  PROC DrawPart187()
    MoveL Offs(pOrigin,194.96,273.17,0.00),v40,fine,tPen\WObj:=wPaper;
    MoveL Offs(pOrigin,194.96,273.17,6.00),v60,z5,tPen\WObj:=wPaper;
    MoveL Offs(pOrigin,203.82,260.21,6.00),vTravel,z5,tPen\WObj:=wPaper;
    MoveL Offs(pOrigin,203.82,260.21,0.00),v60,z0,tPen\WObj:=wPaper;
    MoveL Offs(pOrigin,203.82,257.24,0.00),v40,fine,tPen\WObj:=wPaper;
    MoveL Offs(pOrigin,203.82,257.24,6.00),v60,z5,tPen\WObj:=wPaper;
    MoveL Offs(pOrigin,201.29,252.96,6.00),vTravel,z5,tPen\WObj:=wPaper;
    MoveL Offs(pOrigin,201.29,252.96,0.00),v60,z0,tPen\WObj:=wPaper;
    MoveL Offs(pOrigin,202.04,252.21,0.00),v40,fine,tPen\WObj:=wPaper;
    MoveL Offs(pOrigin,202.04,252.21,6.00),v60,z5,tPen\WObj:=wPaper;
    MoveL Offs(pOrigin,200.69,252.06,6.00),vTravel,z5,tPen\WObj:=wPaper;
    MoveL Offs(pOrigin,200.69,252.06,0.00),v60,z0,tPen\WObj:=wPaper;
    MoveL Offs(pOrigin,202.19,250.56,0.00),v40,fine,tPen\WObj:=wPaper;
    MoveL Offs(pOrigin,202.19,250.56,6.00),v60,z5,tPen\WObj:=wPaper;
    MoveL Offs(pOrigin,197.73,250.01,6.00),vTravel,z5,tPen\WObj:=wPaper;
    MoveL Offs(pOrigin,197.73,250.01,0.00),v60,z0,tPen\WObj:=wPaper;
    MoveL Offs(pOrigin,197.51,250.44,0.00),v40,z0,tPen\WObj:=wPaper;
    MoveL Offs(pOrigin,197.73,250.01,0.00),v40,fine,tPen\WObj:=wPaper;
    MoveL Offs(pOrigin,197.73,250.01,6.00),v60,z5,tPen\WObj:=wPaper;
    MoveL Offs(pOrigin,204.73,243.86,6.00),vTravel,z5,tPen\WObj:=wPaper;
    MoveL Offs(pOrigin,204.73,243.86,0.00),v60,z0,tPen\WObj:=wPaper;
    MoveL Offs(pOrigin,205.94,245.06,0.00),v40,fine,tPen\WObj:=wPaper;
    MoveL Offs(pOrigin,205.94,245.06,6.00),v60,z5,tPen\WObj:=wPaper;
    MoveL Offs(pOrigin,206.28,237.51,6.00),vTravel,z5,tPen\WObj:=wPaper;
    MoveL Offs(pOrigin,206.28,237.51,0.00),v60,z0,tPen\WObj:=wPaper;
    MoveL Offs(pOrigin,208.08,235.71,0.00),v40,fine,tPen\WObj:=wPaper;
    MoveL Offs(pOrigin,208.08,235.71,6.00),v60,z5,tPen\WObj:=wPaper;
    MoveL Offs(pOrigin,203.68,228.55,6.00),vTravel,z5,tPen\WObj:=wPaper;
    MoveL Offs(pOrigin,203.68,228.55,0.00),v60,z0,tPen\WObj:=wPaper;
    MoveL Offs(pOrigin,203.25,229.19,0.00),v40,z0,tPen\WObj:=wPaper;
    MoveL Offs(pOrigin,203.68,228.55,0.00),v40,fine,tPen\WObj:=wPaper;
    MoveL Offs(pOrigin,203.68,228.55,6.00),v60,z5,tPen\WObj:=wPaper;
    MoveL Offs(pOrigin,208.42,223.43,6.00),vTravel,z5,tPen\WObj:=wPaper;
    MoveL Offs(pOrigin,208.42,223.43,0.00),v60,z0,tPen\WObj:=wPaper;
    MoveL Offs(pOrigin,233.21,198.63,0.00),v40,z0,tPen\WObj:=wPaper;
    MoveL Offs(pOrigin,233.51,199.45,0.00),v40,z0,tPen\WObj:=wPaper;
    MoveL Offs(pOrigin,234.26,200.21,0.00),v40,fine,tPen\WObj:=wPaper;
    MoveL Offs(pOrigin,234.26,200.21,6.00),v60,z5,tPen\WObj:=wPaper;
    MoveL Offs(pOrigin,231.26,198.70,6.00),vTravel,z5,tPen\WObj:=wPaper;
    MoveL Offs(pOrigin,231.26,198.70,0.00),v60,z0,tPen\WObj:=wPaper;
    MoveL Offs(pOrigin,229.31,196.74,0.00),v40,z0,tPen\WObj:=wPaper;
    MoveL Offs(pOrigin,230.22,197.10,0.00),v40,z0,tPen\WObj:=wPaper;
    MoveL Offs(pOrigin,230.22,198.16,0.00),v40,z0,tPen\WObj:=wPaper;
    MoveL Offs(pOrigin,231.09,197.95,0.00),v40,z0,tPen\WObj:=wPaper;
    MoveL Offs(pOrigin,230.02,199.01,0.00),v40,z0,tPen\WObj:=wPaper;
    MoveL Offs(pOrigin,231.09,197.95,0.00),v40,fine,tPen\WObj:=wPaper;
    MoveL Offs(pOrigin,231.09,197.95,6.00),v60,z5,tPen\WObj:=wPaper;
    MoveL Offs(pOrigin,229.60,199.65,6.00),vTravel,z5,tPen\WObj:=wPaper;
    MoveL Offs(pOrigin,229.60,199.65,0.00),v60,z0,tPen\WObj:=wPaper;
    MoveL Offs(pOrigin,229.18,200.29,0.00),v40,z0,tPen\WObj:=wPaper;
    MoveL Offs(pOrigin,229.60,199.65,0.00),v40,z0,tPen\WObj:=wPaper;
    MoveL Offs(pOrigin,229.60,199.80,0.00),v40,z0,tPen\WObj:=wPaper;
    MoveL Offs(pOrigin,228.11,199.80,0.00),v40,z0,tPen\WObj:=wPaper;
    MoveL Offs(pOrigin,228.11,199.65,0.00),v40,z0,tPen\WObj:=wPaper;
    MoveL Offs(pOrigin,227.69,200.29,0.00),v40,z0,tPen\WObj:=wPaper;
    MoveL Offs(pOrigin,228.11,199.65,0.00),v40,z0,tPen\WObj:=wPaper;
    MoveL Offs(pOrigin,227.82,199.74,0.00),v40,z0,tPen\WObj:=wPaper;
    MoveL Offs(pOrigin,230.82,202.74,0.00),v40,z0,tPen\WObj:=wPaper;
    MoveL Offs(pOrigin,229.78,203.19,0.00),v40,z0,tPen\WObj:=wPaper;
    MoveL Offs(pOrigin,227.07,200.48,0.00),v40,z0,tPen\WObj:=wPaper;
    MoveL Offs(pOrigin,227.48,200.71,0.00),v40,z0,tPen\WObj:=wPaper;
    MoveL Offs(pOrigin,227.05,201.35,0.00),v40,z0,tPen\WObj:=wPaper;
    MoveL Offs(pOrigin,227.48,200.71,0.00),v40,z0,tPen\WObj:=wPaper;
    MoveL Offs(pOrigin,227.69,200.86,0.00),v40,z0,tPen\WObj:=wPaper;
    MoveL Offs(pOrigin,228.96,200.86,0.00),v40,fine,tPen\WObj:=wPaper;
    MoveL Offs(pOrigin,228.96,200.86,6.00),v60,z5,tPen\WObj:=wPaper;
    MoveL Offs(pOrigin,230.02,201.91,6.00),vTravel,z5,tPen\WObj:=wPaper;
    MoveL Offs(pOrigin,230.02,201.91,0.00),v60,z0,tPen\WObj:=wPaper;
    MoveL Offs(pOrigin,226.84,201.91,0.00),v40,z0,tPen\WObj:=wPaper;
    MoveL Offs(pOrigin,227.05,202.41,0.00),v40,z0,tPen\WObj:=wPaper;
    MoveL Offs(pOrigin,227.05,204.11,0.00),v40,z0,tPen\WObj:=wPaper;
    MoveL Offs(pOrigin,227.90,204.11,0.00),v40,z0,tPen\WObj:=wPaper;
    MoveL Offs(pOrigin,227.05,204.96,0.00),v40,z0,tPen\WObj:=wPaper;
    MoveL Offs(pOrigin,227.90,204.11,0.00),v40,z0,tPen\WObj:=wPaper;
    MoveL Offs(pOrigin,228.11,204.02,0.00),v40,z0,tPen\WObj:=wPaper;
    MoveL Offs(pOrigin,225.56,204.02,0.00),v40,z0,tPen\WObj:=wPaper;
    MoveL Offs(pOrigin,225.77,203.69,0.00),v40,z0,tPen\WObj:=wPaper;
    MoveL Offs(pOrigin,225.56,204.11,0.00),v40,z0,tPen\WObj:=wPaper;
    MoveL Offs(pOrigin,225.77,203.69,0.00),v40,z0,tPen\WObj:=wPaper;
    MoveL Offs(pOrigin,226.00,203.90,0.00),v40,z0,tPen\WObj:=wPaper;
    MoveL Offs(pOrigin,226.00,204.96,0.00),v40,z0,tPen\WObj:=wPaper;
    MoveL Offs(pOrigin,226.13,205.74,0.00),v40,z0,tPen\WObj:=wPaper;
    MoveL Offs(pOrigin,222.80,209.00,0.00),v40,z0,tPen\WObj:=wPaper;
    MoveL Offs(pOrigin,226.13,205.74,0.00),v40,z0,tPen\WObj:=wPaper;
    MoveL Offs(pOrigin,226.64,206.02,0.00),v40,z0,tPen\WObj:=wPaper;
    MoveL Offs(pOrigin,224.99,204.37,0.00),v40,z0,tPen\WObj:=wPaper;
    MoveL Offs(pOrigin,225.14,204.75,0.00),v40,z0,tPen\WObj:=wPaper;
    MoveL Offs(pOrigin,224.71,205.39,0.00),v40,z0,tPen\WObj:=wPaper;
    MoveL Offs(pOrigin,225.14,204.75,0.00),v40,z0,tPen\WObj:=wPaper;
    MoveL Offs(pOrigin,224.92,205.08,0.00),v40,z0,tPen\WObj:=wPaper;
    MoveL Offs(pOrigin,226.84,205.08,0.00),v40,z0,tPen\WObj:=wPaper;
    MoveL Offs(pOrigin,227.39,205.28,0.00),v40,z0,tPen\WObj:=wPaper;
    MoveL Offs(pOrigin,225.43,203.32,0.00),v40,fine,tPen\WObj:=wPaper;
    MoveL Offs(pOrigin,225.43,203.32,6.00),v60,z5,tPen\WObj:=wPaper;
    MoveL Offs(pOrigin,225.71,201.65,6.00),vTravel,z5,tPen\WObj:=wPaper;
    MoveL Offs(pOrigin,225.71,201.65,0.00),v60,z0,tPen\WObj:=wPaper;
    MoveL Offs(pOrigin,236.83,190.53,0.00),v40,z0,tPen\WObj:=wPaper;
    MoveL Offs(pOrigin,236.33,190.33,0.00),v40,z0,tPen\WObj:=wPaper;
    MoveL Offs(pOrigin,233.02,187.02,0.00),v40,z0,tPen\WObj:=wPaper;
    MoveL Offs(pOrigin,233.85,187.32,0.00),v40,z0,tPen\WObj:=wPaper;
    MoveL Offs(pOrigin,236.19,184.99,0.00),v40,z0,tPen\WObj:=wPaper;
    MoveL Offs(pOrigin,237.18,183.50,0.00),v40,z0,tPen\WObj:=wPaper;
    MoveL Offs(pOrigin,237.46,182.23,0.00),v40,z0,tPen\WObj:=wPaper;
    MoveL Offs(pOrigin,237.46,182.23,0.00),v40,z0,tPen\WObj:=wPaper;
    MoveL Offs(pOrigin,238.95,179.25,0.00),v40,z0,tPen\WObj:=wPaper;
    MoveL Offs(pOrigin,238.88,177.55,0.00),v40,z0,tPen\WObj:=wPaper;
    MoveL Offs(pOrigin,238.10,176.91,0.00),v40,z0,tPen\WObj:=wPaper;
    MoveL Offs(pOrigin,237.04,177.05,0.00),v40,z0,tPen\WObj:=wPaper;
    MoveL Offs(pOrigin,236.19,177.76,0.00),v40,z0,tPen\WObj:=wPaper;
    MoveL Offs(pOrigin,235.98,178.61,0.00),v40,z0,tPen\WObj:=wPaper;
    MoveL Offs(pOrigin,235.98,178.61,0.00),v40,z0,tPen\WObj:=wPaper;
    MoveL Offs(pOrigin,235.48,179.04,0.00),v40,z0,tPen\WObj:=wPaper;
    MoveL Offs(pOrigin,235.12,180.10,0.00),v40,z0,tPen\WObj:=wPaper;
    MoveL Offs(pOrigin,235.27,181.59,0.00),v40,z0,tPen\WObj:=wPaper;
    MoveL Offs(pOrigin,236.19,182.23,0.00),v40,z0,tPen\WObj:=wPaper;
    MoveL Offs(pOrigin,237.46,182.23,0.00),v40,fine,tPen\WObj:=wPaper;
    MoveL Offs(pOrigin,237.46,182.23,6.00),v60,z5,tPen\WObj:=wPaper;
    MoveL Offs(pOrigin,236.76,183.29,6.00),vTravel,z5,tPen\WObj:=wPaper;
    MoveL Offs(pOrigin,236.76,183.29,0.00),v60,z0,tPen\WObj:=wPaper;
    MoveL Offs(pOrigin,240.21,186.74,0.00),v40,z0,tPen\WObj:=wPaper;
  ENDPROC

  PROC DrawPart188()
    MoveL Offs(pOrigin,239.80,186.07,0.00),v40,z0,tPen\WObj:=wPaper;
    MoveL Offs(pOrigin,237.04,186.07,0.00),v40,z0,tPen\WObj:=wPaper;
    MoveL Offs(pOrigin,236.82,186.69,0.00),v40,z0,tPen\WObj:=wPaper;
    MoveL Offs(pOrigin,235.98,187.75,0.00),v40,z0,tPen\WObj:=wPaper;
    MoveL Offs(pOrigin,236.82,186.69,0.00),v40,z0,tPen\WObj:=wPaper;
    MoveL Offs(pOrigin,236.40,187.13,0.00),v40,z0,tPen\WObj:=wPaper;
    MoveL Offs(pOrigin,238.95,187.13,0.00),v40,z0,tPen\WObj:=wPaper;
    MoveL Offs(pOrigin,239.31,187.34,0.00),v40,z0,tPen\WObj:=wPaper;
    MoveL Offs(pOrigin,236.61,184.63,0.00),v40,z0,tPen\WObj:=wPaper;
    MoveL Offs(pOrigin,235.86,185.38,0.00),v40,z0,tPen\WObj:=wPaper;
    MoveL Offs(pOrigin,238.57,188.09,0.00),v40,z0,tPen\WObj:=wPaper;
    MoveL Offs(pOrigin,239.24,188.13,0.00),v40,z0,tPen\WObj:=wPaper;
    MoveL Offs(pOrigin,243.74,183.62,0.00),v40,fine,tPen\WObj:=wPaper;
    MoveL Offs(pOrigin,243.74,183.62,6.00),v60,z5,tPen\WObj:=wPaper;
    MoveL Offs(pOrigin,241.80,184.08,6.00),vTravel,z5,tPen\WObj:=wPaper;
    MoveL Offs(pOrigin,241.80,184.08,0.00),v60,z0,tPen\WObj:=wPaper;
    MoveL Offs(pOrigin,227.97,197.90,0.00),v40,fine,tPen\WObj:=wPaper;
    MoveL Offs(pOrigin,227.97,197.90,6.00),v60,z5,tPen\WObj:=wPaper;
    MoveL Offs(pOrigin,230.66,195.58,6.00),vTravel,z5,tPen\WObj:=wPaper;
    MoveL Offs(pOrigin,230.66,195.58,0.00),v60,z0,tPen\WObj:=wPaper;
    MoveL Offs(pOrigin,233.21,195.58,0.00),v40,z0,tPen\WObj:=wPaper;
    MoveL Offs(pOrigin,233.35,196.31,0.00),v40,z0,tPen\WObj:=wPaper;
    MoveL Offs(pOrigin,231.10,194.05,0.00),v40,z0,tPen\WObj:=wPaper;
    MoveL Offs(pOrigin,231.30,194.52,0.00),v40,z0,tPen\WObj:=wPaper;
    MoveL Offs(pOrigin,234.06,194.52,0.00),v40,z0,tPen\WObj:=wPaper;
    MoveL Offs(pOrigin,233.43,194.55,0.00),v40,z0,tPen\WObj:=wPaper;
    MoveL Offs(pOrigin,233.57,193.49,0.00),v40,z0,tPen\WObj:=wPaper;
    MoveL Offs(pOrigin,235.98,190.09,0.00),v40,z0,tPen\WObj:=wPaper;
    MoveL Offs(pOrigin,237.46,188.39,0.00),v40,z0,tPen\WObj:=wPaper;
    MoveL Offs(pOrigin,239.09,187.25,0.00),v40,z0,tPen\WObj:=wPaper;
    MoveL Offs(pOrigin,239.59,186.33,0.00),v40,z0,tPen\WObj:=wPaper;
    MoveL Offs(pOrigin,244.90,184.35,0.00),v40,z0,tPen\WObj:=wPaper;
    MoveL Offs(pOrigin,247.88,183.71,0.00),v40,z0,tPen\WObj:=wPaper;
    MoveL Offs(pOrigin,248.73,183.93,0.00),v40,fine,tPen\WObj:=wPaper;
    MoveL Offs(pOrigin,248.73,183.93,6.00),v60,z5,tPen\WObj:=wPaper;
    MoveL Offs(pOrigin,247.04,183.31,6.00),vTravel,z5,tPen\WObj:=wPaper;
    MoveL Offs(pOrigin,247.04,183.31,0.00),v60,z0,tPen\WObj:=wPaper;
    MoveL Offs(pOrigin,245.24,185.11,0.00),v40,fine,tPen\WObj:=wPaper;
    MoveL Offs(pOrigin,245.24,185.11,6.00),v60,z5,tPen\WObj:=wPaper;
    MoveL Offs(pOrigin,245.69,183.16,6.00),vTravel,z5,tPen\WObj:=wPaper;
    MoveL Offs(pOrigin,245.69,183.16,0.00),v60,z0,tPen\WObj:=wPaper;
    MoveL Offs(pOrigin,242.84,186.02,0.00),v40,z0,tPen\WObj:=wPaper;
    MoveL Offs(pOrigin,242.16,185.70,0.00),v40,z0,tPen\WObj:=wPaper;
    MoveL Offs(pOrigin,241.40,184.95,0.00),v40,z0,tPen\WObj:=wPaper;
    MoveL Offs(pOrigin,240.65,184.20,0.00),v40,z0,tPen\WObj:=wPaper;
    MoveL Offs(pOrigin,237.05,180.59,0.00),v40,z0,tPen\WObj:=wPaper;
    MoveL Offs(pOrigin,237.64,179.69,0.00),v40,z0,tPen\WObj:=wPaper;
    MoveL Offs(pOrigin,241.10,183.15,0.00),v40,z0,tPen\WObj:=wPaper;
    MoveL Offs(pOrigin,240.65,182.86,0.00),v40,z0,tPen\WObj:=wPaper;
    MoveL Offs(pOrigin,240.44,183.29,0.00),v40,z0,tPen\WObj:=wPaper;
    MoveL Offs(pOrigin,240.65,182.86,0.00),v40,z0,tPen\WObj:=wPaper;
    MoveL Offs(pOrigin,240.44,182.90,0.00),v40,z0,tPen\WObj:=wPaper;
    MoveL Offs(pOrigin,239.38,182.90,0.00),v40,z0,tPen\WObj:=wPaper;
    MoveL Offs(pOrigin,239.16,183.07,0.00),v40,z0,tPen\WObj:=wPaper;
    MoveL Offs(pOrigin,238.74,183.71,0.00),v40,z0,tPen\WObj:=wPaper;
    MoveL Offs(pOrigin,239.16,183.07,0.00),v40,z0,tPen\WObj:=wPaper;
    MoveL Offs(pOrigin,238.52,183.96,0.00),v40,z0,tPen\WObj:=wPaper;
    MoveL Offs(pOrigin,240.01,183.96,0.00),v40,z0,tPen\WObj:=wPaper;
    MoveL Offs(pOrigin,239.80,185.02,0.00),v40,z0,tPen\WObj:=wPaper;
    MoveL Offs(pOrigin,237.89,185.02,0.00),v40,z0,tPen\WObj:=wPaper;
    MoveL Offs(pOrigin,238.10,184.77,0.00),v40,z0,tPen\WObj:=wPaper;
    MoveL Offs(pOrigin,237.68,185.41,0.00),v40,z0,tPen\WObj:=wPaper;
    MoveL Offs(pOrigin,238.10,184.77,0.00),v40,z0,tPen\WObj:=wPaper;
    MoveL Offs(pOrigin,238.67,185.41,0.00),v40,z0,tPen\WObj:=wPaper;
    MoveL Offs(pOrigin,238.67,186.69,0.00),v40,z0,tPen\WObj:=wPaper;
    MoveL Offs(pOrigin,239.38,186.26,0.00),v40,z0,tPen\WObj:=wPaper;
    MoveL Offs(pOrigin,239.30,185.41,0.00),v40,z0,tPen\WObj:=wPaper;
    MoveL Offs(pOrigin,242.35,180.74,0.00),v40,z0,tPen\WObj:=wPaper;
    MoveL Offs(pOrigin,245.54,179.39,0.00),v40,z0,tPen\WObj:=wPaper;
    MoveL Offs(pOrigin,247.24,179.04,0.00),v40,fine,tPen\WObj:=wPaper;
    MoveL Offs(pOrigin,247.24,179.04,6.00),v60,z5,tPen\WObj:=wPaper;
    MoveL Offs(pOrigin,245.41,178.97,6.00),vTravel,z5,tPen\WObj:=wPaper;
    MoveL Offs(pOrigin,245.41,178.97,0.00),v60,z0,tPen\WObj:=wPaper;
    MoveL Offs(pOrigin,230.08,194.30,0.00),v40,fine,tPen\WObj:=wPaper;
    MoveL Offs(pOrigin,230.08,194.30,6.00),v60,z5,tPen\WObj:=wPaper;
    MoveL Offs(pOrigin,231.69,193.16,6.00),vTravel,z5,tPen\WObj:=wPaper;
    MoveL Offs(pOrigin,231.69,193.16,0.00),v60,z0,tPen\WObj:=wPaper;
    MoveL Offs(pOrigin,234.10,195.56,0.00),v40,z0,tPen\WObj:=wPaper;
    MoveL Offs(pOrigin,234.57,195.78,0.00),v40,z0,tPen\WObj:=wPaper;
    MoveL Offs(pOrigin,239.83,190.52,0.00),v40,fine,tPen\WObj:=wPaper;
    MoveL Offs(pOrigin,239.83,190.52,6.00),v60,z5,tPen\WObj:=wPaper;
    MoveL Offs(pOrigin,241.63,190.22,6.00),vTravel,z5,tPen\WObj:=wPaper;
    MoveL Offs(pOrigin,241.63,190.22,0.00),v60,z0,tPen\WObj:=wPaper;
    MoveL Offs(pOrigin,238.17,193.67,0.00),v40,fine,tPen\WObj:=wPaper;
    MoveL Offs(pOrigin,238.17,193.67,6.00),v60,z5,tPen\WObj:=wPaper;
    MoveL Offs(pOrigin,236.79,193.77,6.00),vTravel,z5,tPen\WObj:=wPaper;
    MoveL Offs(pOrigin,236.79,193.77,0.00),v60,z0,tPen\WObj:=wPaper;
    MoveL Offs(pOrigin,233.48,190.47,0.00),v40,z0,tPen\WObj:=wPaper;
    MoveL Offs(pOrigin,234.06,190.30,0.00),v40,z0,tPen\WObj:=wPaper;
    MoveL Offs(pOrigin,233.43,191.15,0.00),v40,z0,tPen\WObj:=wPaper;
    MoveL Offs(pOrigin,234.06,190.30,0.00),v40,z0,tPen\WObj:=wPaper;
    MoveL Offs(pOrigin,234.28,190.30,0.00),v40,z0,tPen\WObj:=wPaper;
    MoveL Offs(pOrigin,235.76,190.30,0.00),v40,z0,tPen\WObj:=wPaper;
    MoveL Offs(pOrigin,235.76,190.09,0.00),v40,z0,tPen\WObj:=wPaper;
    MoveL Offs(pOrigin,235.34,190.73,0.00),v40,z0,tPen\WObj:=wPaper;
    MoveL Offs(pOrigin,235.76,190.09,0.00),v40,z0,tPen\WObj:=wPaper;
    MoveL Offs(pOrigin,235.58,191.07,0.00),v40,z0,tPen\WObj:=wPaper;
    MoveL Offs(pOrigin,234.08,189.57,0.00),v40,z0,tPen\WObj:=wPaper;
    MoveL Offs(pOrigin,234.91,189.24,0.00),v40,z0,tPen\WObj:=wPaper;
    MoveL Offs(pOrigin,236.40,189.24,0.00),v40,z0,tPen\WObj:=wPaper;
    MoveL Offs(pOrigin,236.92,189.43,0.00),v40,z0,tPen\WObj:=wPaper;
    MoveL Offs(pOrigin,234.07,186.57,0.00),v40,z0,tPen\WObj:=wPaper;
    MoveL Offs(pOrigin,234.97,185.98,0.00),v40,z0,tPen\WObj:=wPaper;
    MoveL Offs(pOrigin,237.67,188.68,0.00),v40,z0,tPen\WObj:=wPaper;
    MoveL Offs(pOrigin,237.46,188.18,0.00),v40,z0,tPen\WObj:=wPaper;
    MoveL Offs(pOrigin,235.55,188.18,0.00),v40,fine,tPen\WObj:=wPaper;
    MoveL Offs(pOrigin,235.55,188.18,6.00),v60,z5,tPen\WObj:=wPaper;
    MoveL Offs(pOrigin,237.04,188.60,6.00),vTravel,z5,tPen\WObj:=wPaper;
    MoveL Offs(pOrigin,237.04,188.60,0.00),v60,z0,tPen\WObj:=wPaper;
    MoveL Offs(pOrigin,236.40,189.24,0.00),v40,z0,tPen\WObj:=wPaper;
    MoveL Offs(pOrigin,237.04,188.60,0.00),v40,fine,tPen\WObj:=wPaper;
    MoveL Offs(pOrigin,237.04,188.60,6.00),v60,z5,tPen\WObj:=wPaper;
    MoveL Offs(pOrigin,237.61,187.54,6.00),vTravel,z5,tPen\WObj:=wPaper;
    MoveL Offs(pOrigin,237.61,187.54,0.00),v60,z0,tPen\WObj:=wPaper;
    MoveL Offs(pOrigin,237.61,186.48,0.00),v40,fine,tPen\WObj:=wPaper;
    MoveL Offs(pOrigin,237.61,186.48,6.00),v60,z5,tPen\WObj:=wPaper;
    MoveL Offs(pOrigin,241.26,186.30,6.00),vTravel,z5,tPen\WObj:=wPaper;
    MoveL Offs(pOrigin,241.26,186.30,0.00),v60,z0,tPen\WObj:=wPaper;
    MoveL Offs(pOrigin,236.15,181.19,0.00),v40,fine,tPen\WObj:=wPaper;
    MoveL Offs(pOrigin,236.15,181.19,6.00),v60,z5,tPen\WObj:=wPaper;
  ENDPROC

  PROC DrawPart189()
    MoveL Offs(pOrigin,238.09,178.65,6.00),vTravel,z5,tPen\WObj:=wPaper;
    MoveL Offs(pOrigin,238.09,178.65,0.00),v60,z0,tPen\WObj:=wPaper;
    MoveL Offs(pOrigin,239.14,179.70,0.00),v40,z0,tPen\WObj:=wPaper;
    MoveL Offs(pOrigin,239.89,180.45,0.00),v40,z0,tPen\WObj:=wPaper;
    MoveL Offs(pOrigin,241.70,182.25,0.00),v40,z0,tPen\WObj:=wPaper;
    MoveL Offs(pOrigin,241.29,181.85,0.00),v40,z0,tPen\WObj:=wPaper;
    MoveL Offs(pOrigin,240.01,181.85,0.00),v40,z0,tPen\WObj:=wPaper;
    MoveL Offs(pOrigin,239.80,182.01,0.00),v40,z0,tPen\WObj:=wPaper;
    MoveL Offs(pOrigin,239.38,182.65,0.00),v40,z0,tPen\WObj:=wPaper;
    MoveL Offs(pOrigin,239.80,182.01,0.00),v40,fine,tPen\WObj:=wPaper;
    MoveL Offs(pOrigin,239.80,182.01,6.00),v60,z5,tPen\WObj:=wPaper;
    MoveL Offs(pOrigin,240.44,180.79,6.00),vTravel,z5,tPen\WObj:=wPaper;
    MoveL Offs(pOrigin,240.44,180.79,0.00),v60,z0,tPen\WObj:=wPaper;
    MoveL Offs(pOrigin,242.14,180.79,0.00),v40,z0,tPen\WObj:=wPaper;
    MoveL Offs(pOrigin,242.35,180.52,0.00),v40,z0,tPen\WObj:=wPaper;
    MoveL Offs(pOrigin,245.25,171.60,0.00),v40,z0,tPen\WObj:=wPaper;
    MoveL Offs(pOrigin,245.96,170.32,0.00),v40,z0,tPen\WObj:=wPaper;
    MoveL Offs(pOrigin,248.80,167.85,0.00),v40,z0,tPen\WObj:=wPaper;
    MoveL Offs(pOrigin,248.30,168.20,0.00),v40,z0,tPen\WObj:=wPaper;
    MoveL Offs(pOrigin,248.09,168.12,0.00),v40,z0,tPen\WObj:=wPaper;
    MoveL Offs(pOrigin,246.60,168.12,0.00),v40,z0,tPen\WObj:=wPaper;
    MoveL Offs(pOrigin,246.44,167.59,0.00),v40,z0,tPen\WObj:=wPaper;
    MoveL Offs(pOrigin,247.95,169.09,0.00),v40,z0,tPen\WObj:=wPaper;
    MoveL Offs(pOrigin,247.88,168.41,0.00),v40,z0,tPen\WObj:=wPaper;
    MoveL Offs(pOrigin,247.45,168.84,0.00),v40,z0,tPen\WObj:=wPaper;
    MoveL Offs(pOrigin,247.88,168.41,0.00),v40,z0,tPen\WObj:=wPaper;
    MoveL Offs(pOrigin,248.84,168.49,0.00),v40,z0,tPen\WObj:=wPaper;
    MoveL Offs(pOrigin,247.34,166.99,0.00),v40,z0,tPen\WObj:=wPaper;
    MoveL Offs(pOrigin,248.09,167.06,0.00),v40,z0,tPen\WObj:=wPaper;
    MoveL Offs(pOrigin,249.58,167.06,0.00),v40,z0,tPen\WObj:=wPaper;
    MoveL Offs(pOrigin,249.36,167.56,0.00),v40,z0,tPen\WObj:=wPaper;
    MoveL Offs(pOrigin,252.76,164.66,0.00),v40,z0,tPen\WObj:=wPaper;
    MoveL Offs(pOrigin,253.40,164.59,0.00),v40,z0,tPen\WObj:=wPaper;
    MoveL Offs(pOrigin,258.08,168.84,0.00),v40,z0,tPen\WObj:=wPaper;
    MoveL Offs(pOrigin,259.00,170.32,0.00),v40,z0,tPen\WObj:=wPaper;
    MoveL Offs(pOrigin,259.77,173.94,0.00),v40,z0,tPen\WObj:=wPaper;
    MoveL Offs(pOrigin,260.98,176.49,0.00),v40,z0,tPen\WObj:=wPaper;
    MoveL Offs(pOrigin,261.12,177.55,0.00),v40,z0,tPen\WObj:=wPaper;
    MoveL Offs(pOrigin,263.39,180.10,0.00),v40,z0,tPen\WObj:=wPaper;
    MoveL Offs(pOrigin,267.85,186.48,0.00),v40,z0,tPen\WObj:=wPaper;
    MoveL Offs(pOrigin,268.27,188.18,0.00),v40,z0,tPen\WObj:=wPaper;
    MoveL Offs(pOrigin,268.27,188.18,0.00),v40,z0,tPen\WObj:=wPaper;
    MoveL Offs(pOrigin,270.61,188.18,0.00),v40,fine,tPen\WObj:=wPaper;
    MoveL Offs(pOrigin,270.61,188.18,6.00),v60,z5,tPen\WObj:=wPaper;
    MoveL Offs(pOrigin,273.59,188.18,6.00),vTravel,z5,tPen\WObj:=wPaper;
    MoveL Offs(pOrigin,273.59,188.18,0.00),v60,z0,tPen\WObj:=wPaper;
    MoveL Offs(pOrigin,275.71,188.18,0.00),v40,z0,tPen\WObj:=wPaper;
    MoveL Offs(pOrigin,276.47,188.65,0.00),v40,z0,tPen\WObj:=wPaper;
    MoveL Offs(pOrigin,274.97,187.15,0.00),v40,z0,tPen\WObj:=wPaper;
    MoveL Offs(pOrigin,275.71,187.13,0.00),v40,z0,tPen\WObj:=wPaper;
    MoveL Offs(pOrigin,276.99,187.13,0.00),v40,z0,tPen\WObj:=wPaper;
    MoveL Offs(pOrigin,277.07,187.75,0.00),v40,z0,tPen\WObj:=wPaper;
    MoveL Offs(pOrigin,275.71,186.40,0.00),v40,z0,tPen\WObj:=wPaper;
    MoveL Offs(pOrigin,276.14,186.48,0.00),v40,z0,tPen\WObj:=wPaper;
    MoveL Offs(pOrigin,275.71,187.11,0.00),v40,z0,tPen\WObj:=wPaper;
    MoveL Offs(pOrigin,276.14,186.48,0.00),v40,z0,tPen\WObj:=wPaper;
    MoveL Offs(pOrigin,276.35,186.07,0.00),v40,z0,tPen\WObj:=wPaper;
    MoveL Offs(pOrigin,277.41,186.07,0.00),v40,z0,tPen\WObj:=wPaper;
    MoveL Offs(pOrigin,277.66,186.86,0.00),v40,z0,tPen\WObj:=wPaper;
    MoveL Offs(pOrigin,276.16,185.35,0.00),v40,fine,tPen\WObj:=wPaper;
    MoveL Offs(pOrigin,276.16,185.35,6.00),v60,z5,tPen\WObj:=wPaper;
    MoveL Offs(pOrigin,278.40,184.61,6.00),vTravel,z5,tPen\WObj:=wPaper;
    MoveL Offs(pOrigin,278.40,184.61,0.00),v60,z0,tPen\WObj:=wPaper;
    MoveL Offs(pOrigin,276.60,182.81,0.00),v40,z0,tPen\WObj:=wPaper;
    MoveL Offs(pOrigin,276.25,182.47,0.00),v40,z0,tPen\WObj:=wPaper;
    MoveL Offs(pOrigin,282.57,176.16,0.00),v40,fine,tPen\WObj:=wPaper;
    MoveL Offs(pOrigin,282.57,176.16,6.00),v60,z5,tPen\WObj:=wPaper;
    MoveL Offs(pOrigin,282.27,174.96,6.00),vTravel,z5,tPen\WObj:=wPaper;
    MoveL Offs(pOrigin,282.27,174.96,0.00),v60,z0,tPen\WObj:=wPaper;
    MoveL Offs(pOrigin,275.66,181.57,0.00),v40,z0,tPen\WObj:=wPaper;
    MoveL Offs(pOrigin,276.30,181.01,0.00),v40,z0,tPen\WObj:=wPaper;
    MoveL Offs(pOrigin,278.85,183.56,0.00),v40,z0,tPen\WObj:=wPaper;
    MoveL Offs(pOrigin,279.25,183.96,0.00),v40,z0,tPen\WObj:=wPaper;
    MoveL Offs(pOrigin,268.28,194.93,0.00),v40,z0,tPen\WObj:=wPaper;
    MoveL Offs(pOrigin,269.17,195.53,0.00),v40,z0,tPen\WObj:=wPaper;
    MoveL Offs(pOrigin,273.38,191.32,0.00),v40,z0,tPen\WObj:=wPaper;
    MoveL Offs(pOrigin,274.13,192.07,0.00),v40,z0,tPen\WObj:=wPaper;
    MoveL Offs(pOrigin,270.22,195.97,0.00),v40,z0,tPen\WObj:=wPaper;
    MoveL Offs(pOrigin,269.90,195.52,0.00),v40,z0,tPen\WObj:=wPaper;
    MoveL Offs(pOrigin,267.04,192.67,0.00),v40,z0,tPen\WObj:=wPaper;
    MoveL Offs(pOrigin,266.79,191.94,0.00),v40,z0,tPen\WObj:=wPaper;
    MoveL Offs(pOrigin,265.29,193.44,0.00),v40,z0,tPen\WObj:=wPaper;
    MoveL Offs(pOrigin,264.24,192.99,0.00),v40,z0,tPen\WObj:=wPaper;
    MoveL Offs(pOrigin,265.74,191.49,0.00),v40,z0,tPen\WObj:=wPaper;
    MoveL Offs(pOrigin,264.79,191.91,0.00),v40,z0,tPen\WObj:=wPaper;
    MoveL Offs(pOrigin,266.45,193.56,0.00),v40,z0,tPen\WObj:=wPaper;
    MoveL Offs(pOrigin,266.33,193.89,0.00),v40,z0,tPen\WObj:=wPaper;
    MoveL Offs(pOrigin,267.84,192.38,0.00),v40,z0,tPen\WObj:=wPaper;
    MoveL Offs(pOrigin,268.88,192.83,0.00),v40,z0,tPen\WObj:=wPaper;
    MoveL Offs(pOrigin,267.23,194.48,0.00),v40,fine,tPen\WObj:=wPaper;
    MoveL Offs(pOrigin,267.23,194.48,6.00),v60,z5,tPen\WObj:=wPaper;
    MoveL Offs(pOrigin,270.04,194.17,6.00),vTravel,z5,tPen\WObj:=wPaper;
    MoveL Offs(pOrigin,270.04,194.17,0.00),v60,z0,tPen\WObj:=wPaper;
    MoveL Offs(pOrigin,281.46,205.59,0.00),v40,z0,tPen\WObj:=wPaper;
    MoveL Offs(pOrigin,281.24,205.81,0.00),v40,z0,tPen\WObj:=wPaper;
    MoveL Offs(pOrigin,281.45,206.24,0.00),v40,z0,tPen\WObj:=wPaper;
    MoveL Offs(pOrigin,281.24,205.81,0.00),v40,z0,tPen\WObj:=wPaper;
    MoveL Offs(pOrigin,281.24,206.14,0.00),v40,z0,tPen\WObj:=wPaper;
    MoveL Offs(pOrigin,278.90,206.14,0.00),v40,z0,tPen\WObj:=wPaper;
    MoveL Offs(pOrigin,278.62,207.23,0.00),v40,z0,tPen\WObj:=wPaper;
    MoveL Offs(pOrigin,285.69,214.29,0.00),v40,z0,tPen\WObj:=wPaper;
    MoveL Offs(pOrigin,286.34,214.20,0.00),v40,z0,tPen\WObj:=wPaper;
    MoveL Offs(pOrigin,281.69,218.86,0.00),v40,z0,tPen\WObj:=wPaper;
    MoveL Offs(pOrigin,282.28,219.75,0.00),v40,z0,tPen\WObj:=wPaper;
    MoveL Offs(pOrigin,286.79,215.25,0.00),v40,fine,tPen\WObj:=wPaper;
    MoveL Offs(pOrigin,286.79,215.25,6.00),v60,z5,tPen\WObj:=wPaper;
    MoveL Offs(pOrigin,285.75,213.30,6.00),vTravel,z5,tPen\WObj:=wPaper;
    MoveL Offs(pOrigin,285.75,213.30,0.00),v60,z0,tPen\WObj:=wPaper;
    MoveL Offs(pOrigin,283.49,215.56,0.00),v40,z0,tPen\WObj:=wPaper;
    MoveL Offs(pOrigin,283.89,215.49,0.00),v40,z0,tPen\WObj:=wPaper;
    MoveL Offs(pOrigin,292.01,223.60,0.00),v40,fine,tPen\WObj:=wPaper;
    MoveL Offs(pOrigin,292.01,223.60,6.00),v60,z5,tPen\WObj:=wPaper;
    MoveL Offs(pOrigin,290.59,224.94,6.00),vTravel,z5,tPen\WObj:=wPaper;
    MoveL Offs(pOrigin,290.59,224.94,0.00),v60,z0,tPen\WObj:=wPaper;
    MoveL Offs(pOrigin,290.80,224.51,0.00),v40,z0,tPen\WObj:=wPaper;
    MoveL Offs(pOrigin,290.59,224.94,0.00),v40,z0,tPen\WObj:=wPaper;
    MoveL Offs(pOrigin,290.66,225.25,0.00),v40,z0,tPen\WObj:=wPaper;
    MoveL Offs(pOrigin,284.20,218.78,0.00),v40,z0,tPen\WObj:=wPaper;
    MoveL Offs(pOrigin,283.36,219.41,0.00),v40,z0,tPen\WObj:=wPaper;
    MoveL Offs(pOrigin,280.81,215.59,0.00),v40,z0,tPen\WObj:=wPaper;
  ENDPROC

  PROC DrawPart190()
    MoveL Offs(pOrigin,278.90,213.89,0.00),v40,fine,tPen\WObj:=wPaper;
    MoveL Offs(pOrigin,278.90,213.89,6.00),v60,z5,tPen\WObj:=wPaper;
    MoveL Offs(pOrigin,278.05,211.55,6.00),vTravel,z5,tPen\WObj:=wPaper;
    MoveL Offs(pOrigin,278.05,211.55,0.00),v60,z0,tPen\WObj:=wPaper;
    MoveL Offs(pOrigin,274.65,208.15,0.00),v40,z0,tPen\WObj:=wPaper;
    MoveL Offs(pOrigin,270.40,204.75,0.00),v40,fine,tPen\WObj:=wPaper;
    MoveL Offs(pOrigin,270.40,204.75,6.00),v60,z5,tPen\WObj:=wPaper;
    MoveL Offs(pOrigin,276.66,202.28,6.00),vTravel,z5,tPen\WObj:=wPaper;
    MoveL Offs(pOrigin,276.66,202.28,0.00),v60,z0,tPen\WObj:=wPaper;
    MoveL Offs(pOrigin,282.82,208.44,0.00),v40,z0,tPen\WObj:=wPaper;
    MoveL Offs(pOrigin,282.51,208.36,0.00),v40,z0,tPen\WObj:=wPaper;
    MoveL Offs(pOrigin,282.73,208.79,0.00),v40,z0,tPen\WObj:=wPaper;
    MoveL Offs(pOrigin,282.51,208.36,0.00),v40,z0,tPen\WObj:=wPaper;
    MoveL Offs(pOrigin,282.30,208.25,0.00),v40,z0,tPen\WObj:=wPaper;
    MoveL Offs(pOrigin,280.39,208.25,0.00),v40,z0,tPen\WObj:=wPaper;
    MoveL Offs(pOrigin,280.91,208.36,0.00),v40,z0,tPen\WObj:=wPaper;
    MoveL Offs(pOrigin,280.91,206.66,0.00),v40,z0,tPen\WObj:=wPaper;
    MoveL Offs(pOrigin,281.88,207.19,0.00),v40,z0,tPen\WObj:=wPaper;
    MoveL Offs(pOrigin,279.54,207.19,0.00),v40,z0,tPen\WObj:=wPaper;
    MoveL Offs(pOrigin,279.85,207.09,0.00),v40,z0,tPen\WObj:=wPaper;
    MoveL Offs(pOrigin,279.85,205.18,0.00),v40,z0,tPen\WObj:=wPaper;
    MoveL Offs(pOrigin,280.60,205.08,0.00),v40,z0,tPen\WObj:=wPaper;
    MoveL Offs(pOrigin,278.26,205.08,0.00),v40,fine,tPen\WObj:=wPaper;
    MoveL Offs(pOrigin,278.26,205.08,6.00),v60,z5,tPen\WObj:=wPaper;
    MoveL Offs(pOrigin,278.05,202.97,6.00),vTravel,z5,tPen\WObj:=wPaper;
    MoveL Offs(pOrigin,278.05,202.97,0.00),v60,z0,tPen\WObj:=wPaper;
    MoveL Offs(pOrigin,279.54,202.97,0.00),v40,fine,tPen\WObj:=wPaper;
    MoveL Offs(pOrigin,279.54,202.97,6.00),v60,z5,tPen\WObj:=wPaper;
    MoveL Offs(pOrigin,278.05,202.62,6.00),vTravel,z5,tPen\WObj:=wPaper;
    MoveL Offs(pOrigin,278.05,202.62,0.00),v60,z0,tPen\WObj:=wPaper;
    MoveL Offs(pOrigin,278.26,203.05,0.00),v40,z0,tPen\WObj:=wPaper;
    MoveL Offs(pOrigin,278.05,202.62,0.00),v40,fine,tPen\WObj:=wPaper;
    MoveL Offs(pOrigin,278.05,202.62,6.00),v60,z5,tPen\WObj:=wPaper;
    MoveL Offs(pOrigin,280.39,204.32,6.00),vTravel,z5,tPen\WObj:=wPaper;
    MoveL Offs(pOrigin,280.39,204.32,0.00),v60,z0,tPen\WObj:=wPaper;
    MoveL Offs(pOrigin,280.60,204.75,0.00),v40,z0,tPen\WObj:=wPaper;
    MoveL Offs(pOrigin,280.39,204.32,0.00),v40,z0,tPen\WObj:=wPaper;
    MoveL Offs(pOrigin,280.81,204.96,0.00),v40,z0,tPen\WObj:=wPaper;
    MoveL Offs(pOrigin,281.02,205.39,0.00),v40,z0,tPen\WObj:=wPaper;
    MoveL Offs(pOrigin,280.81,204.96,0.00),v40,z0,tPen\WObj:=wPaper;
    MoveL Offs(pOrigin,281.28,204.33,0.00),v40,z0,tPen\WObj:=wPaper;
    MoveL Offs(pOrigin,278.28,207.33,0.00),v40,z0,tPen\WObj:=wPaper;
    MoveL Offs(pOrigin,279.02,208.08,0.00),v40,z0,tPen\WObj:=wPaper;
    MoveL Offs(pOrigin,281.73,205.37,0.00),v40,z0,tPen\WObj:=wPaper;
    MoveL Offs(pOrigin,282.32,206.27,0.00),v40,z0,tPen\WObj:=wPaper;
    MoveL Offs(pOrigin,279.77,208.83,0.00),v40,z0,tPen\WObj:=wPaper;
    MoveL Offs(pOrigin,280.21,209.87,0.00),v40,z0,tPen\WObj:=wPaper;
    MoveL Offs(pOrigin,282.77,207.32,0.00),v40,z0,tPen\WObj:=wPaper;
    MoveL Offs(pOrigin,282.09,207.51,0.00),v40,z0,tPen\WObj:=wPaper;
    MoveL Offs(pOrigin,282.30,207.94,0.00),v40,z0,tPen\WObj:=wPaper;
    MoveL Offs(pOrigin,282.09,207.51,0.00),v40,fine,tPen\WObj:=wPaper;
    MoveL Offs(pOrigin,282.09,207.51,6.00),v60,z5,tPen\WObj:=wPaper;
    MoveL Offs(pOrigin,283.22,208.37,6.00),vTravel,z5,tPen\WObj:=wPaper;
    MoveL Offs(pOrigin,283.22,208.37,0.00),v60,z0,tPen\WObj:=wPaper;
    MoveL Offs(pOrigin,280.81,210.77,0.00),v40,z0,tPen\WObj:=wPaper;
    MoveL Offs(pOrigin,281.56,211.52,0.00),v40,z0,tPen\WObj:=wPaper;
    MoveL Offs(pOrigin,283.81,209.26,0.00),v40,z0,tPen\WObj:=wPaper;
    MoveL Offs(pOrigin,282.94,209.30,0.00),v40,z0,tPen\WObj:=wPaper;
    MoveL Offs(pOrigin,281.24,209.30,0.00),v40,z0,tPen\WObj:=wPaper;
    MoveL Offs(pOrigin,281.66,209.85,0.00),v40,z0,tPen\WObj:=wPaper;
    MoveL Offs(pOrigin,282.09,210.49,0.00),v40,z0,tPen\WObj:=wPaper;
    MoveL Offs(pOrigin,281.66,209.85,0.00),v40,z0,tPen\WObj:=wPaper;
    MoveL Offs(pOrigin,282.09,210.36,0.00),v40,z0,tPen\WObj:=wPaper;
    MoveL Offs(pOrigin,283.36,210.36,0.00),v40,z0,tPen\WObj:=wPaper;
    MoveL Offs(pOrigin,283.36,210.06,0.00),v40,z0,tPen\WObj:=wPaper;
    MoveL Offs(pOrigin,283.58,210.49,0.00),v40,z0,tPen\WObj:=wPaper;
    MoveL Offs(pOrigin,283.36,210.06,0.00),v40,fine,tPen\WObj:=wPaper;
    MoveL Offs(pOrigin,283.36,210.06,6.00),v60,z5,tPen\WObj:=wPaper;
    MoveL Offs(pOrigin,282.30,210.91,6.00),vTravel,z5,tPen\WObj:=wPaper;
    MoveL Offs(pOrigin,282.30,210.91,0.00),v60,z0,tPen\WObj:=wPaper;
    MoveL Offs(pOrigin,282.51,211.34,0.00),v40,z0,tPen\WObj:=wPaper;
    MoveL Offs(pOrigin,282.30,210.91,0.00),v40,z0,tPen\WObj:=wPaper;
    MoveL Offs(pOrigin,282.73,211.42,0.00),v40,z0,tPen\WObj:=wPaper;
    MoveL Offs(pOrigin,283.79,211.42,0.00),v40,z0,tPen\WObj:=wPaper;
    MoveL Offs(pOrigin,284.21,212.47,0.00),v40,z0,tPen\WObj:=wPaper;
    MoveL Offs(pOrigin,283.15,212.47,0.00),v40,z0,tPen\WObj:=wPaper;
    MoveL Offs(pOrigin,283.15,212.61,0.00),v40,z0,tPen\WObj:=wPaper;
    MoveL Offs(pOrigin,283.36,213.04,0.00),v40,z0,tPen\WObj:=wPaper;
    MoveL Offs(pOrigin,283.15,212.61,0.00),v40,z0,tPen\WObj:=wPaper;
    MoveL Offs(pOrigin,283.79,213.53,0.00),v40,z0,tPen\WObj:=wPaper;
    MoveL Offs(pOrigin,284.85,213.53,0.00),v40,fine,tPen\WObj:=wPaper;
    MoveL Offs(pOrigin,284.85,213.53,6.00),v60,z5,tPen\WObj:=wPaper;
    MoveL Offs(pOrigin,285.30,212.25,6.00),vTravel,z5,tPen\WObj:=wPaper;
    MoveL Offs(pOrigin,285.30,212.25,0.00),v60,z0,tPen\WObj:=wPaper;
    MoveL Offs(pOrigin,283.05,214.51,0.00),v40,fine,tPen\WObj:=wPaper;
    MoveL Offs(pOrigin,283.05,214.51,6.00),v60,z5,tPen\WObj:=wPaper;
    MoveL Offs(pOrigin,278.99,218.56,6.00),vTravel,z5,tPen\WObj:=wPaper;
    MoveL Offs(pOrigin,278.99,218.56,0.00),v60,z0,tPen\WObj:=wPaper;
    MoveL Offs(pOrigin,277.94,219.62,0.00),v40,z0,tPen\WObj:=wPaper;
    MoveL Offs(pOrigin,277.19,218.87,0.00),v40,z0,tPen\WObj:=wPaper;
    MoveL Offs(pOrigin,278.24,217.82,0.00),v40,z0,tPen\WObj:=wPaper;
    MoveL Offs(pOrigin,277.50,217.07,0.00),v40,z0,tPen\WObj:=wPaper;
    MoveL Offs(pOrigin,276.44,218.12,0.00),v40,z0,tPen\WObj:=wPaper;
    MoveL Offs(pOrigin,275.70,217.38,0.00),v40,z0,tPen\WObj:=wPaper;
    MoveL Offs(pOrigin,276.75,216.32,0.00),v40,z0,tPen\WObj:=wPaper;
    MoveL Offs(pOrigin,276.00,215.58,0.00),v40,z0,tPen\WObj:=wPaper;
    MoveL Offs(pOrigin,274.80,216.78,0.00),v40,z0,tPen\WObj:=wPaper;
    MoveL Offs(pOrigin,274.05,216.03,0.00),v40,z0,tPen\WObj:=wPaper;
    MoveL Offs(pOrigin,274.96,215.13,0.00),v40,z0,tPen\WObj:=wPaper;
    MoveL Offs(pOrigin,274.06,214.54,0.00),v40,z0,tPen\WObj:=wPaper;
    MoveL Offs(pOrigin,273.31,215.29,0.00),v40,fine,tPen\WObj:=wPaper;
    MoveL Offs(pOrigin,273.31,215.29,6.00),v60,z5,tPen\WObj:=wPaper;
    MoveL Offs(pOrigin,270.19,217.93,6.00),vTravel,z5,tPen\WObj:=wPaper;
    MoveL Offs(pOrigin,270.19,217.93,0.00),v60,z0,tPen\WObj:=wPaper;
    MoveL Offs(pOrigin,268.98,216.44,0.00),v40,z0,tPen\WObj:=wPaper;
    MoveL Offs(pOrigin,268.84,215.80,0.00),v40,z0,tPen\WObj:=wPaper;
    MoveL Offs(pOrigin,267.64,215.38,0.00),v40,z0,tPen\WObj:=wPaper;
    MoveL Offs(pOrigin,267.64,215.38,0.00),v40,z0,tPen\WObj:=wPaper;
    MoveL Offs(pOrigin,267.85,216.44,0.00),v40,z0,tPen\WObj:=wPaper;
    MoveL Offs(pOrigin,269.12,216.86,0.00),v40,fine,tPen\WObj:=wPaper;
    MoveL Offs(pOrigin,269.12,216.86,6.00),v60,z5,tPen\WObj:=wPaper;
    MoveL Offs(pOrigin,267.76,216.35,6.00),vTravel,z5,tPen\WObj:=wPaper;
    MoveL Offs(pOrigin,267.76,216.35,0.00),v60,z0,tPen\WObj:=wPaper;
    MoveL Offs(pOrigin,268.66,215.45,0.00),v40,z0,tPen\WObj:=wPaper;
    MoveL Offs(pOrigin,267.64,215.38,0.00),v40,z0,tPen\WObj:=wPaper;
    MoveL Offs(pOrigin,265.51,213.46,0.00),v40,z0,tPen\WObj:=wPaper;
    MoveL Offs(pOrigin,265.51,213.46,0.00),v40,z0,tPen\WObj:=wPaper;
    MoveL Offs(pOrigin,264.45,212.40,0.00),v40,fine,tPen\WObj:=wPaper;
    MoveL Offs(pOrigin,264.45,212.40,6.00),v60,z5,tPen\WObj:=wPaper;
    MoveL Offs(pOrigin,268.49,212.40,6.00),vTravel,z5,tPen\WObj:=wPaper;
  ENDPROC

  PROC DrawPart191()
    MoveL Offs(pOrigin,268.49,212.40,0.00),v60,z0,tPen\WObj:=wPaper;
    MoveL Offs(pOrigin,273.38,214.88,0.00),v40,z0,tPen\WObj:=wPaper;
    MoveL Offs(pOrigin,276.99,217.50,0.00),v40,z0,tPen\WObj:=wPaper;
    MoveL Offs(pOrigin,279.75,220.26,0.00),v40,z0,tPen\WObj:=wPaper;
    MoveL Offs(pOrigin,282.51,224.30,0.00),v40,fine,tPen\WObj:=wPaper;
    MoveL Offs(pOrigin,282.51,224.30,6.00),v60,z5,tPen\WObj:=wPaper;
    MoveL Offs(pOrigin,282.88,220.65,6.00),vTravel,z5,tPen\WObj:=wPaper;
    MoveL Offs(pOrigin,282.88,220.65,0.00),v60,z0,tPen\WObj:=wPaper;
    MoveL Offs(pOrigin,290.54,212.99,0.00),v40,fine,tPen\WObj:=wPaper;
    MoveL Offs(pOrigin,290.54,212.99,6.00),v60,z5,tPen\WObj:=wPaper;
    MoveL Offs(pOrigin,294.68,217.32,6.00),vTravel,z5,tPen\WObj:=wPaper;
    MoveL Offs(pOrigin,294.68,217.32,0.00),v60,z0,tPen\WObj:=wPaper;
    MoveL Offs(pOrigin,296.03,218.67,0.00),v40,z0,tPen\WObj:=wPaper;
    MoveL Offs(pOrigin,296.11,218.35,0.00),v40,z0,tPen\WObj:=wPaper;
    MoveL Offs(pOrigin,296.33,217.93,0.00),v40,z0,tPen\WObj:=wPaper;
    MoveL Offs(pOrigin,296.11,218.35,0.00),v40,z0,tPen\WObj:=wPaper;
    MoveL Offs(pOrigin,296.32,217.75,0.00),v40,z0,tPen\WObj:=wPaper;
    MoveL Offs(pOrigin,294.84,217.75,0.00),v40,z0,tPen\WObj:=wPaper;
    MoveL Offs(pOrigin,294.09,218.22,0.00),v40,z0,tPen\WObj:=wPaper;
    MoveL Offs(pOrigin,295.44,219.57,0.00),v40,z0,tPen\WObj:=wPaper;
    MoveL Offs(pOrigin,295.05,219.62,0.00),v40,z0,tPen\WObj:=wPaper;
    MoveL Offs(pOrigin,295.26,219.20,0.00),v40,z0,tPen\WObj:=wPaper;
    MoveL Offs(pOrigin,295.05,219.62,0.00),v40,z0,tPen\WObj:=wPaper;
    MoveL Offs(pOrigin,294.69,220.31,0.00),v40,z0,tPen\WObj:=wPaper;
    MoveL Offs(pOrigin,293.19,218.81,0.00),v40,z0,tPen\WObj:=wPaper;
    MoveL Offs(pOrigin,293.77,218.77,0.00),v40,z0,tPen\WObj:=wPaper;
    MoveL Offs(pOrigin,292.92,219.62,0.00),v40,z0,tPen\WObj:=wPaper;
    MoveL Offs(pOrigin,293.77,218.77,0.00),v40,z0,tPen\WObj:=wPaper;
    MoveL Offs(pOrigin,293.99,218.81,0.00),v40,z0,tPen\WObj:=wPaper;
    MoveL Offs(pOrigin,295.26,218.81,0.00),v40,fine,tPen\WObj:=wPaper;
    MoveL Offs(pOrigin,295.26,218.81,6.00),v60,z5,tPen\WObj:=wPaper;
    MoveL Offs(pOrigin,294.20,219.86,6.00),vTravel,z5,tPen\WObj:=wPaper;
    MoveL Offs(pOrigin,294.20,219.86,0.00),v60,z0,tPen\WObj:=wPaper;
    MoveL Offs(pOrigin,293.14,219.86,0.00),v40,z0,tPen\WObj:=wPaper;
    MoveL Offs(pOrigin,292.59,219.71,0.00),v40,z0,tPen\WObj:=wPaper;
    MoveL Offs(pOrigin,293.94,221.06,0.00),v40,z0,tPen\WObj:=wPaper;
    MoveL Offs(pOrigin,293.56,221.11,0.00),v40,z0,tPen\WObj:=wPaper;
    MoveL Offs(pOrigin,293.35,221.54,0.00),v40,z0,tPen\WObj:=wPaper;
    MoveL Offs(pOrigin,293.56,221.11,0.00),v40,z0,tPen\WObj:=wPaper;
    MoveL Offs(pOrigin,293.35,220.92,0.00),v40,z0,tPen\WObj:=wPaper;
    MoveL Offs(pOrigin,292.08,220.92,0.00),v40,z0,tPen\WObj:=wPaper;
    MoveL Offs(pOrigin,291.65,221.32,0.00),v40,z0,tPen\WObj:=wPaper;
    MoveL Offs(pOrigin,291.01,221.96,0.00),v40,z0,tPen\WObj:=wPaper;
    MoveL Offs(pOrigin,291.65,221.32,0.00),v40,fine,tPen\WObj:=wPaper;
    MoveL Offs(pOrigin,291.65,221.32,6.00),v60,z5,tPen\WObj:=wPaper;
    MoveL Offs(pOrigin,292.50,220.26,6.00),vTravel,z5,tPen\WObj:=wPaper;
    MoveL Offs(pOrigin,292.50,220.26,0.00),v60,z0,tPen\WObj:=wPaper;
    MoveL Offs(pOrigin,292.08,220.69,0.00),v40,z0,tPen\WObj:=wPaper;
    MoveL Offs(pOrigin,292.50,220.26,0.00),v40,fine,tPen\WObj:=wPaper;
    MoveL Offs(pOrigin,292.50,220.26,6.00),v60,z5,tPen\WObj:=wPaper;
    MoveL Offs(pOrigin,294.41,220.26,6.00),vTravel,z5,tPen\WObj:=wPaper;
    MoveL Offs(pOrigin,294.41,220.26,0.00),v60,z0,tPen\WObj:=wPaper;
    MoveL Offs(pOrigin,294.62,219.84,0.00),v40,z0,tPen\WObj:=wPaper;
    MoveL Offs(pOrigin,294.41,220.26,0.00),v40,fine,tPen\WObj:=wPaper;
    MoveL Offs(pOrigin,294.41,220.26,6.00),v60,z5,tPen\WObj:=wPaper;
    MoveL Offs(pOrigin,296.93,218.07,6.00),vTravel,z5,tPen\WObj:=wPaper;
    MoveL Offs(pOrigin,296.93,218.07,0.00),v60,z0,tPen\WObj:=wPaper;
    MoveL Offs(pOrigin,295.43,216.57,0.00),v40,z0,tPen\WObj:=wPaper;
    MoveL Offs(pOrigin,295.90,216.70,0.00),v40,z0,tPen\WObj:=wPaper;
    MoveL Offs(pOrigin,297.39,216.70,0.00),v40,z0,tPen\WObj:=wPaper;
    MoveL Offs(pOrigin,297.39,217.07,0.00),v40,z0,tPen\WObj:=wPaper;
    MoveL Offs(pOrigin,297.60,216.65,0.00),v40,z0,tPen\WObj:=wPaper;
    MoveL Offs(pOrigin,297.39,217.07,0.00),v40,z0,tPen\WObj:=wPaper;
    MoveL Offs(pOrigin,297.53,217.18,0.00),v40,z0,tPen\WObj:=wPaper;
    MoveL Offs(pOrigin,296.18,215.82,0.00),v40,z0,tPen\WObj:=wPaper;
    MoveL Offs(pOrigin,296.96,215.64,0.00),v40,z0,tPen\WObj:=wPaper;
    MoveL Offs(pOrigin,298.45,215.64,0.00),v40,z0,tPen\WObj:=wPaper;
    MoveL Offs(pOrigin,298.88,215.80,0.00),v40,z0,tPen\WObj:=wPaper;
    MoveL Offs(pOrigin,299.09,215.38,0.00),v40,z0,tPen\WObj:=wPaper;
    MoveL Offs(pOrigin,298.88,215.80,0.00),v40,z0,tPen\WObj:=wPaper;
    MoveL Offs(pOrigin,299.17,215.83,0.00),v40,z0,tPen\WObj:=wPaper;
    MoveL Offs(pOrigin,297.67,214.33,0.00),v40,z0,tPen\WObj:=wPaper;
    MoveL Offs(pOrigin,298.02,214.58,0.00),v40,z0,tPen\WObj:=wPaper;
    MoveL Offs(pOrigin,299.51,214.58,0.00),v40,z0,tPen\WObj:=wPaper;
    MoveL Offs(pOrigin,299.73,214.74,0.00),v40,z0,tPen\WObj:=wPaper;
    MoveL Offs(pOrigin,299.51,215.16,0.00),v40,z0,tPen\WObj:=wPaper;
    MoveL Offs(pOrigin,299.73,214.74,0.00),v40,z0,tPen\WObj:=wPaper;
    MoveL Offs(pOrigin,299.92,215.09,0.00),v40,z0,tPen\WObj:=wPaper;
    MoveL Offs(pOrigin,298.42,213.58,0.00),v40,z0,tPen\WObj:=wPaper;
    MoveL Offs(pOrigin,299.02,213.39,0.00),v40,z0,tPen\WObj:=wPaper;
    MoveL Offs(pOrigin,294.20,218.14,0.00),v40,z0,tPen\WObj:=wPaper;
    MoveL Offs(pOrigin,299.02,213.39,0.00),v40,z0,tPen\WObj:=wPaper;
    MoveL Offs(pOrigin,299.09,213.53,0.00),v40,z0,tPen\WObj:=wPaper;
    MoveL Offs(pOrigin,301.00,213.53,0.00),v40,z0,tPen\WObj:=wPaper;
    MoveL Offs(pOrigin,301.71,213.89,0.00),v40,z0,tPen\WObj:=wPaper;
    MoveL Offs(pOrigin,299.91,212.09,0.00),v40,z0,tPen\WObj:=wPaper;
    MoveL Offs(pOrigin,299.94,212.47,0.00),v40,z0,tPen\WObj:=wPaper;
    MoveL Offs(pOrigin,304.40,212.47,0.00),v40,z0,tPen\WObj:=wPaper;
    MoveL Offs(pOrigin,304.11,213.30,0.00),v40,z0,tPen\WObj:=wPaper;
    MoveL Offs(pOrigin,301.25,210.45,0.00),v40,z0,tPen\WObj:=wPaper;
    MoveL Offs(pOrigin,301.42,210.70,0.00),v40,z0,tPen\WObj:=wPaper;
    MoveL Offs(pOrigin,301.00,211.34,0.00),v40,z0,tPen\WObj:=wPaper;
    MoveL Offs(pOrigin,301.42,210.70,0.00),v40,z0,tPen\WObj:=wPaper;
    MoveL Offs(pOrigin,301.85,210.36,0.00),v40,z0,tPen\WObj:=wPaper;
    MoveL Offs(pOrigin,303.76,210.36,0.00),v40,z0,tPen\WObj:=wPaper;
    MoveL Offs(pOrigin,304.19,209.85,0.00),v40,z0,tPen\WObj:=wPaper;
    MoveL Offs(pOrigin,303.98,210.27,0.00),v40,z0,tPen\WObj:=wPaper;
    MoveL Offs(pOrigin,304.19,209.85,0.00),v40,z0,tPen\WObj:=wPaper;
    MoveL Offs(pOrigin,304.40,209.30,0.00),v40,z0,tPen\WObj:=wPaper;
    MoveL Offs(pOrigin,302.91,209.30,0.00),v40,z0,tPen\WObj:=wPaper;
    MoveL Offs(pOrigin,302.75,208.95,0.00),v40,z0,tPen\WObj:=wPaper;
    MoveL Offs(pOrigin,306.65,212.86,0.00),v40,z0,tPen\WObj:=wPaper;
    MoveL Offs(pOrigin,307.02,212.94,0.00),v40,z0,tPen\WObj:=wPaper;
    MoveL Offs(pOrigin,311.53,208.43,0.00),v40,z0,tPen\WObj:=wPaper;
    MoveL Offs(pOrigin,312.05,209.30,0.00),v40,z0,tPen\WObj:=wPaper;
    MoveL Offs(pOrigin,315.24,209.30,0.00),v40,z0,tPen\WObj:=wPaper;
    MoveL Offs(pOrigin,315.24,208.25,0.00),v40,z0,tPen\WObj:=wPaper;
    MoveL Offs(pOrigin,318.21,208.25,0.00),v40,z0,tPen\WObj:=wPaper;
    MoveL Offs(pOrigin,318.92,208.70,0.00),v40,z0,tPen\WObj:=wPaper;
    MoveL Offs(pOrigin,317.27,207.05,0.00),v40,z0,tPen\WObj:=wPaper;
    MoveL Offs(pOrigin,318.21,207.19,0.00),v40,z0,tPen\WObj:=wPaper;
    MoveL Offs(pOrigin,320.98,207.19,0.00),v40,z0,tPen\WObj:=wPaper;
    MoveL Offs(pOrigin,321.02,207.81,0.00),v40,z0,tPen\WObj:=wPaper;
    MoveL Offs(pOrigin,319.52,206.31,0.00),v40,z0,tPen\WObj:=wPaper;
    MoveL Offs(pOrigin,320.56,205.86,0.00),v40,z0,tPen\WObj:=wPaper;
    MoveL Offs(pOrigin,322.07,207.37,0.00),v40,fine,tPen\WObj:=wPaper;
    MoveL Offs(pOrigin,322.07,207.37,6.00),v60,z5,tPen\WObj:=wPaper;
    MoveL Offs(pOrigin,323.31,206.66,6.00),vTravel,z5,tPen\WObj:=wPaper;
    MoveL Offs(pOrigin,323.31,206.66,0.00),v60,z0,tPen\WObj:=wPaper;
    MoveL Offs(pOrigin,323.74,206.45,0.00),v40,z0,tPen\WObj:=wPaper;
  ENDPROC

  PROC DrawPart192()
    MoveL Offs(pOrigin,323.31,206.66,0.00),v40,z0,tPen\WObj:=wPaper;
    MoveL Offs(pOrigin,323.52,206.14,0.00),v40,z0,tPen\WObj:=wPaper;
    MoveL Offs(pOrigin,320.98,206.14,0.00),v40,fine,tPen\WObj:=wPaper;
    MoveL Offs(pOrigin,320.98,206.14,6.00),v60,z5,tPen\WObj:=wPaper;
    MoveL Offs(pOrigin,322.66,204.97,6.00),vTravel,z5,tPen\WObj:=wPaper;
    MoveL Offs(pOrigin,322.66,204.97,0.00),v60,z0,tPen\WObj:=wPaper;
    MoveL Offs(pOrigin,324.31,206.62,0.00),v40,fine,tPen\WObj:=wPaper;
    MoveL Offs(pOrigin,324.31,206.62,6.00),v60,z5,tPen\WObj:=wPaper;
    MoveL Offs(pOrigin,323.68,203.75,6.00),vTravel,z5,tPen\WObj:=wPaper;
    MoveL Offs(pOrigin,323.68,203.75,0.00),v60,z0,tPen\WObj:=wPaper;
    MoveL Offs(pOrigin,318.12,209.31,0.00),v40,z0,tPen\WObj:=wPaper;
    MoveL Offs(pOrigin,317.73,209.00,0.00),v40,z0,tPen\WObj:=wPaper;
    MoveL Offs(pOrigin,316.22,207.50,0.00),v40,z0,tPen\WObj:=wPaper;
    MoveL Offs(pOrigin,316.18,206.77,0.00),v40,z0,tPen\WObj:=wPaper;
    MoveL Offs(pOrigin,311.22,211.73,0.00),v40,z0,tPen\WObj:=wPaper;
    MoveL Offs(pOrigin,311.14,211.38,0.00),v40,z0,tPen\WObj:=wPaper;
    MoveL Offs(pOrigin,309.49,209.72,0.00),v40,z0,tPen\WObj:=wPaper;
    MoveL Offs(pOrigin,309.43,209.03,0.00),v40,z0,tPen\WObj:=wPaper;
    MoveL Offs(pOrigin,305.07,213.39,0.00),v40,z0,tPen\WObj:=wPaper;
    MoveL Offs(pOrigin,305.30,213.01,0.00),v40,z0,tPen\WObj:=wPaper;
    MoveL Offs(pOrigin,302.00,209.70,0.00),v40,z0,tPen\WObj:=wPaper;
    MoveL Offs(pOrigin,302.49,209.64,0.00),v40,z0,tPen\WObj:=wPaper;
    MoveL Offs(pOrigin,301.85,210.27,0.00),v40,z0,tPen\WObj:=wPaper;
    MoveL Offs(pOrigin,302.49,209.64,0.00),v40,fine,tPen\WObj:=wPaper;
    MoveL Offs(pOrigin,302.49,209.64,6.00),v60,z5,tPen\WObj:=wPaper;
    MoveL Offs(pOrigin,302.03,211.12,6.00),vTravel,z5,tPen\WObj:=wPaper;
    MoveL Offs(pOrigin,302.03,211.12,0.00),v60,z0,tPen\WObj:=wPaper;
    MoveL Offs(pOrigin,302.03,212.82,0.00),v40,z0,tPen\WObj:=wPaper;
    MoveL Offs(pOrigin,303.09,212.40,0.00),v40,z0,tPen\WObj:=wPaper;
    MoveL Offs(pOrigin,303.09,211.12,0.00),v40,fine,tPen\WObj:=wPaper;
    MoveL Offs(pOrigin,303.09,211.12,6.00),v60,z5,tPen\WObj:=wPaper;
    MoveL Offs(pOrigin,305.00,209.71,6.00),vTravel,z5,tPen\WObj:=wPaper;
    MoveL Offs(pOrigin,305.00,209.71,0.00),v60,z0,tPen\WObj:=wPaper;
    MoveL Offs(pOrigin,303.34,208.06,0.00),v40,z0,tPen\WObj:=wPaper;
    MoveL Offs(pOrigin,303.55,208.15,0.00),v40,z0,tPen\WObj:=wPaper;
    MoveL Offs(pOrigin,303.12,208.79,0.00),v40,z0,tPen\WObj:=wPaper;
    MoveL Offs(pOrigin,303.55,208.15,0.00),v40,z0,tPen\WObj:=wPaper;
    MoveL Offs(pOrigin,303.76,208.25,0.00),v40,z0,tPen\WObj:=wPaper;
    MoveL Offs(pOrigin,305.25,208.25,0.00),v40,z0,tPen\WObj:=wPaper;
    MoveL Offs(pOrigin,305.44,208.66,0.00),v40,z0,tPen\WObj:=wPaper;
    MoveL Offs(pOrigin,304.09,207.31,0.00),v40,z0,tPen\WObj:=wPaper;
    MoveL Offs(pOrigin,304.40,207.30,0.00),v40,z0,tPen\WObj:=wPaper;
    MoveL Offs(pOrigin,303.76,207.94,0.00),v40,z0,tPen\WObj:=wPaper;
    MoveL Offs(pOrigin,304.40,207.30,0.00),v40,z0,tPen\WObj:=wPaper;
    MoveL Offs(pOrigin,304.61,207.19,0.00),v40,z0,tPen\WObj:=wPaper;
    MoveL Offs(pOrigin,306.10,207.19,0.00),v40,z0,tPen\WObj:=wPaper;
    MoveL Offs(pOrigin,306.52,207.09,0.00),v40,z0,tPen\WObj:=wPaper;
    MoveL Offs(pOrigin,306.74,206.66,0.00),v40,z0,tPen\WObj:=wPaper;
    MoveL Offs(pOrigin,306.52,207.09,0.00),v40,z0,tPen\WObj:=wPaper;
    MoveL Offs(pOrigin,306.93,207.17,0.00),v40,z0,tPen\WObj:=wPaper;
    MoveL Offs(pOrigin,305.43,205.67,0.00),v40,z0,tPen\WObj:=wPaper;
    MoveL Offs(pOrigin,305.67,205.60,0.00),v40,z0,tPen\WObj:=wPaper;
    MoveL Offs(pOrigin,305.25,206.24,0.00),v40,z0,tPen\WObj:=wPaper;
    MoveL Offs(pOrigin,305.67,205.60,0.00),v40,z0,tPen\WObj:=wPaper;
    MoveL Offs(pOrigin,305.46,206.14,0.00),v40,z0,tPen\WObj:=wPaper;
    MoveL Offs(pOrigin,306.95,206.14,0.00),v40,z0,tPen\WObj:=wPaper;
    MoveL Offs(pOrigin,307.53,206.27,0.00),v40,z0,tPen\WObj:=wPaper;
    MoveL Offs(pOrigin,306.03,204.77,0.00),v40,z0,tPen\WObj:=wPaper;
    MoveL Offs(pOrigin,306.31,205.08,0.00),v40,z0,tPen\WObj:=wPaper;
    MoveL Offs(pOrigin,308.44,205.08,0.00),v40,z0,tPen\WObj:=wPaper;
    MoveL Offs(pOrigin,308.37,204.54,0.00),v40,z0,tPen\WObj:=wPaper;
    MoveL Offs(pOrigin,308.37,203.48,0.00),v40,z0,tPen\WObj:=wPaper;
    MoveL Offs(pOrigin,308.01,202.97,0.00),v40,z0,tPen\WObj:=wPaper;
    MoveL Offs(pOrigin,309.71,202.97,0.00),v40,z0,tPen\WObj:=wPaper;
    MoveL Offs(pOrigin,309.71,202.84,0.00),v40,z0,tPen\WObj:=wPaper;
    MoveL Offs(pOrigin,309.50,203.26,0.00),v40,z0,tPen\WObj:=wPaper;
    MoveL Offs(pOrigin,309.71,202.84,0.00),v40,fine,tPen\WObj:=wPaper;
    MoveL Offs(pOrigin,309.71,202.84,6.00),v60,z5,tPen\WObj:=wPaper;
    MoveL Offs(pOrigin,309.92,204.02,6.00),vTravel,z5,tPen\WObj:=wPaper;
    MoveL Offs(pOrigin,309.92,204.02,0.00),v60,z0,tPen\WObj:=wPaper;
    MoveL Offs(pOrigin,307.16,204.02,0.00),v40,z0,tPen\WObj:=wPaper;
    MoveL Offs(pOrigin,306.63,203.87,0.00),v40,z0,tPen\WObj:=wPaper;
    MoveL Offs(pOrigin,308.43,205.68,0.00),v40,z0,tPen\WObj:=wPaper;
    MoveL Offs(pOrigin,307.59,205.60,0.00),v40,z0,tPen\WObj:=wPaper;
    MoveL Offs(pOrigin,307.38,206.02,0.00),v40,z0,tPen\WObj:=wPaper;
    MoveL Offs(pOrigin,307.59,205.60,0.00),v40,fine,tPen\WObj:=wPaper;
    MoveL Offs(pOrigin,307.59,205.60,6.00),v60,z5,tPen\WObj:=wPaper;
    MoveL Offs(pOrigin,309.48,205.23,6.00),vTravel,z5,tPen\WObj:=wPaper;
    MoveL Offs(pOrigin,309.48,205.23,0.00),v60,z0,tPen\WObj:=wPaper;
    MoveL Offs(pOrigin,307.37,203.13,0.00),v40,z0,tPen\WObj:=wPaper;
    MoveL Offs(pOrigin,307.80,203.05,0.00),v40,z0,tPen\WObj:=wPaper;
    MoveL Offs(pOrigin,307.16,203.69,0.00),v40,z0,tPen\WObj:=wPaper;
    MoveL Offs(pOrigin,307.80,203.05,0.00),v40,z0,tPen\WObj:=wPaper;
    MoveL Offs(pOrigin,308.12,202.38,0.00),v40,z0,tPen\WObj:=wPaper;
    MoveL Offs(pOrigin,310.82,205.08,0.00),v40,fine,tPen\WObj:=wPaper;
    MoveL Offs(pOrigin,310.82,205.08,6.00),v60,z5,tPen\WObj:=wPaper;
    MoveL Offs(pOrigin,309.74,205.74,6.00),vTravel,z5,tPen\WObj:=wPaper;
    MoveL Offs(pOrigin,309.74,205.74,0.00),v60,z0,tPen\WObj:=wPaper;
    MoveL Offs(pOrigin,312.89,202.58,0.00),v40,z0,tPen\WObj:=wPaper;
    MoveL Offs(pOrigin,313.21,202.99,0.00),v40,z0,tPen\WObj:=wPaper;
    MoveL Offs(pOrigin,314.57,204.35,0.00),v40,z0,tPen\WObj:=wPaper;
    MoveL Offs(pOrigin,315.43,204.52,0.00),v40,z0,tPen\WObj:=wPaper;
    MoveL Offs(pOrigin,318.89,201.07,0.00),v40,z0,tPen\WObj:=wPaper;
    MoveL Offs(pOrigin,318.15,201.96,0.00),v40,z0,tPen\WObj:=wPaper;
    MoveL Offs(pOrigin,319.06,202.86,0.00),v40,z0,tPen\WObj:=wPaper;
    MoveL Offs(pOrigin,318.01,203.31,0.00),v40,z0,tPen\WObj:=wPaper;
    MoveL Offs(pOrigin,317.11,202.41,0.00),v40,z0,tPen\WObj:=wPaper;
    MoveL Offs(pOrigin,316.79,201.67,0.00),v40,z0,tPen\WObj:=wPaper;
    MoveL Offs(pOrigin,313.33,205.13,0.00),v40,z0,tPen\WObj:=wPaper;
    MoveL Offs(pOrigin,313.37,204.64,0.00),v40,z0,tPen\WObj:=wPaper;
    MoveL Offs(pOrigin,312.17,203.44,0.00),v40,fine,tPen\WObj:=wPaper;
    MoveL Offs(pOrigin,312.17,203.44,6.00),v60,z5,tPen\WObj:=wPaper;
    MoveL Offs(pOrigin,314.56,202.85,6.00),vTravel,z5,tPen\WObj:=wPaper;
    MoveL Offs(pOrigin,314.56,202.85,0.00),v60,z0,tPen\WObj:=wPaper;
    MoveL Offs(pOrigin,315.76,204.05,0.00),v40,fine,tPen\WObj:=wPaper;
    MoveL Offs(pOrigin,315.76,204.05,6.00),v60,z5,tPen\WObj:=wPaper;
    MoveL Offs(pOrigin,315.18,207.94,6.00),vTravel,z5,tPen\WObj:=wPaper;
    MoveL Offs(pOrigin,315.18,207.94,0.00),v60,z0,tPen\WObj:=wPaper;
    MoveL Offs(pOrigin,316.68,209.45,0.00),v40,fine,tPen\WObj:=wPaper;
    MoveL Offs(pOrigin,316.68,209.45,6.00),v60,z5,tPen\WObj:=wPaper;
    MoveL Offs(pOrigin,314.43,210.19,6.00),vTravel,z5,tPen\WObj:=wPaper;
    MoveL Offs(pOrigin,314.43,210.19,0.00),v60,z0,tPen\WObj:=wPaper;
    MoveL Offs(pOrigin,313.08,208.84,0.00),v40,fine,tPen\WObj:=wPaper;
    MoveL Offs(pOrigin,313.08,208.84,6.00),v60,z5,tPen\WObj:=wPaper;
    MoveL Offs(pOrigin,309.79,211.52,6.00),vTravel,z5,tPen\WObj:=wPaper;
    MoveL Offs(pOrigin,309.79,211.52,0.00),v60,z0,tPen\WObj:=wPaper;
    MoveL Offs(pOrigin,308.29,210.02,0.00),v40,fine,tPen\WObj:=wPaper;
    MoveL Offs(pOrigin,308.29,210.02,6.00),v60,z5,tPen\WObj:=wPaper;
    MoveL Offs(pOrigin,307.55,212.26,6.00),vTravel,z5,tPen\WObj:=wPaper;
    MoveL Offs(pOrigin,307.55,212.26,0.00),v60,z0,tPen\WObj:=wPaper;
  ENDPROC

  PROC DrawPart193()
    MoveL Offs(pOrigin,305.90,210.61,0.00),v40,z0,tPen\WObj:=wPaper;
    MoveL Offs(pOrigin,305.83,209.64,0.00),v40,z0,tPen\WObj:=wPaper;
    MoveL Offs(pOrigin,287.35,228.13,0.00),v40,z0,tPen\WObj:=wPaper;
    MoveL Offs(pOrigin,288.13,228.68,0.00),v40,z0,tPen\WObj:=wPaper;
    MoveL Offs(pOrigin,291.28,231.84,0.00),v40,z0,tPen\WObj:=wPaper;
    MoveL Offs(pOrigin,291.53,231.41,0.00),v40,z0,tPen\WObj:=wPaper;
    MoveL Offs(pOrigin,289.13,233.81,0.00),v40,z0,tPen\WObj:=wPaper;
    MoveL Offs(pOrigin,289.64,233.18,0.00),v40,z0,tPen\WObj:=wPaper;
    MoveL Offs(pOrigin,292.04,235.59,0.00),v40,z0,tPen\WObj:=wPaper;
    MoveL Offs(pOrigin,292.42,235.00,0.00),v40,z0,tPen\WObj:=wPaper;
    MoveL Offs(pOrigin,289.87,237.56,0.00),v40,z0,tPen\WObj:=wPaper;
    MoveL Offs(pOrigin,290.25,238.28,0.00),v40,z0,tPen\WObj:=wPaper;
    MoveL Offs(pOrigin,292.36,240.38,0.00),v40,z0,tPen\WObj:=wPaper;
    MoveL Offs(pOrigin,292.95,239.48,0.00),v40,z0,tPen\WObj:=wPaper;
    MoveL Offs(pOrigin,290.25,236.78,0.00),v40,z0,tPen\WObj:=wPaper;
    MoveL Offs(pOrigin,289.57,236.36,0.00),v40,z0,tPen\WObj:=wPaper;
    MoveL Offs(pOrigin,292.28,233.65,0.00),v40,z0,tPen\WObj:=wPaper;
    MoveL Offs(pOrigin,291.59,233.64,0.00),v40,z0,tPen\WObj:=wPaper;
    MoveL Offs(pOrigin,289.03,231.08,0.00),v40,z0,tPen\WObj:=wPaper;
    MoveL Offs(pOrigin,288.54,231.42,0.00),v40,z0,tPen\WObj:=wPaper;
    MoveL Offs(pOrigin,290.94,229.01,0.00),v40,z0,tPen\WObj:=wPaper;
    MoveL Offs(pOrigin,290.83,229.89,0.00),v40,z0,tPen\WObj:=wPaper;
    MoveL Offs(pOrigin,286.47,225.53,0.00),v40,z0,tPen\WObj:=wPaper;
    MoveL Offs(pOrigin,286.98,225.14,0.00),v40,z0,tPen\WObj:=wPaper;
    MoveL Offs(pOrigin,290.16,225.14,0.00),v40,z0,tPen\WObj:=wPaper;
    MoveL Offs(pOrigin,289.36,225.36,0.00),v40,z0,tPen\WObj:=wPaper;
    MoveL Offs(pOrigin,289.36,223.66,0.00),v40,fine,tPen\WObj:=wPaper;
    MoveL Offs(pOrigin,289.36,223.66,6.00),v60,z5,tPen\WObj:=wPaper;
    MoveL Offs(pOrigin,289.52,221.98,6.00),vTravel,z5,tPen\WObj:=wPaper;
    MoveL Offs(pOrigin,289.52,221.98,0.00),v60,z0,tPen\WObj:=wPaper;
    MoveL Offs(pOrigin,285.70,221.98,0.00),v40,fine,tPen\WObj:=wPaper;
    MoveL Offs(pOrigin,285.70,221.98,6.00),v60,z5,tPen\WObj:=wPaper;
    MoveL Offs(pOrigin,287.25,222.18,6.00),vTravel,z5,tPen\WObj:=wPaper;
    MoveL Offs(pOrigin,287.25,222.18,0.00),v60,z0,tPen\WObj:=wPaper;
    MoveL Offs(pOrigin,287.25,225.15,0.00),v40,z0,tPen\WObj:=wPaper;
    MoveL Offs(pOrigin,287.40,226.00,0.00),v40,z0,tPen\WObj:=wPaper;
    MoveL Offs(pOrigin,287.61,226.43,0.00),v40,z0,tPen\WObj:=wPaper;
    MoveL Offs(pOrigin,287.40,226.00,0.00),v40,z0,tPen\WObj:=wPaper;
    MoveL Offs(pOrigin,286.31,226.18,0.00),v40,z0,tPen\WObj:=wPaper;
    MoveL Offs(pOrigin,317.41,195.08,0.00),v40,fine,tPen\WObj:=wPaper;
    MoveL Offs(pOrigin,317.41,195.08,6.00),v60,z5,tPen\WObj:=wPaper;
    MoveL Offs(pOrigin,318.00,192.43,6.00),vTravel,z5,tPen\WObj:=wPaper;
    MoveL Offs(pOrigin,318.00,192.43,0.00),v60,z0,tPen\WObj:=wPaper;
    MoveL Offs(pOrigin,317.79,192.85,0.00),v40,z0,tPen\WObj:=wPaper;
    MoveL Offs(pOrigin,318.00,192.43,0.00),v40,fine,tPen\WObj:=wPaper;
    MoveL Offs(pOrigin,318.00,192.43,6.00),v60,z5,tPen\WObj:=wPaper;
    MoveL Offs(pOrigin,318.64,191.36,6.00),vTravel,z5,tPen\WObj:=wPaper;
    MoveL Offs(pOrigin,318.64,191.36,0.00),v60,z0,tPen\WObj:=wPaper;
    MoveL Offs(pOrigin,318.42,191.79,0.00),v40,z0,tPen\WObj:=wPaper;
    MoveL Offs(pOrigin,318.64,191.36,0.00),v40,z0,tPen\WObj:=wPaper;
    MoveL Offs(pOrigin,319.82,191.18,0.00),v40,z0,tPen\WObj:=wPaper;
    MoveL Offs(pOrigin,300.29,210.71,0.00),v40,fine,tPen\WObj:=wPaper;
    MoveL Offs(pOrigin,300.29,210.71,6.00),v60,z5,tPen\WObj:=wPaper;
    MoveL Offs(pOrigin,299.16,212.84,6.00),vTravel,z5,tPen\WObj:=wPaper;
    MoveL Offs(pOrigin,299.16,212.84,0.00),v60,z0,tPen\WObj:=wPaper;
    MoveL Offs(pOrigin,300.82,214.49,0.00),v40,z0,tPen\WObj:=wPaper;
    MoveL Offs(pOrigin,300.36,214.10,0.00),v40,z0,tPen\WObj:=wPaper;
    MoveL Offs(pOrigin,300.15,214.52,0.00),v40,z0,tPen\WObj:=wPaper;
    MoveL Offs(pOrigin,300.36,214.10,0.00),v40,fine,tPen\WObj:=wPaper;
    MoveL Offs(pOrigin,300.36,214.10,6.00),v60,z5,tPen\WObj:=wPaper;
    MoveL Offs(pOrigin,298.43,216.58,6.00),vTravel,z5,tPen\WObj:=wPaper;
    MoveL Offs(pOrigin,298.43,216.58,0.00),v60,z0,tPen\WObj:=wPaper;
    MoveL Offs(pOrigin,296.92,215.08,0.00),v40,fine,tPen\WObj:=wPaper;
    MoveL Offs(pOrigin,296.92,215.08,6.00),v60,z5,tPen\WObj:=wPaper;
    MoveL Offs(pOrigin,298.02,216.44,6.00),vTravel,z5,tPen\WObj:=wPaper;
    MoveL Offs(pOrigin,298.02,216.44,0.00),v60,z0,tPen\WObj:=wPaper;
    MoveL Offs(pOrigin,298.45,216.01,0.00),v40,z0,tPen\WObj:=wPaper;
    MoveL Offs(pOrigin,298.02,216.44,0.00),v40,fine,tPen\WObj:=wPaper;
    MoveL Offs(pOrigin,298.02,216.44,6.00),v60,z5,tPen\WObj:=wPaper;
    MoveL Offs(pOrigin,296.75,217.71,6.00),vTravel,z5,tPen\WObj:=wPaper;
    MoveL Offs(pOrigin,296.75,217.71,0.00),v60,z0,tPen\WObj:=wPaper;
    MoveL Offs(pOrigin,296.96,217.29,0.00),v40,z0,tPen\WObj:=wPaper;
    MoveL Offs(pOrigin,296.75,217.71,0.00),v40,fine,tPen\WObj:=wPaper;
    MoveL Offs(pOrigin,296.75,217.71,6.00),v60,z5,tPen\WObj:=wPaper;
    MoveL Offs(pOrigin,290.35,226.62,6.00),vTravel,z5,tPen\WObj:=wPaper;
    MoveL Offs(pOrigin,290.35,226.62,0.00),v60,z0,tPen\WObj:=wPaper;
    MoveL Offs(pOrigin,287.80,229.17,0.00),v40,fine,tPen\WObj:=wPaper;
    MoveL Offs(pOrigin,287.80,229.17,6.00),v60,z5,tPen\WObj:=wPaper;
    MoveL Offs(pOrigin,288.09,230.37,6.00),vTravel,z5,tPen\WObj:=wPaper;
    MoveL Offs(pOrigin,288.09,230.37,0.00),v60,z0,tPen\WObj:=wPaper;
    MoveL Offs(pOrigin,290.50,227.97,0.00),v40,fine,tPen\WObj:=wPaper;
    MoveL Offs(pOrigin,290.50,227.97,6.00),v60,z5,tPen\WObj:=wPaper;
    MoveL Offs(pOrigin,291.39,230.06,6.00),vTravel,z5,tPen\WObj:=wPaper;
    MoveL Offs(pOrigin,291.39,230.06,0.00),v60,z0,tPen\WObj:=wPaper;
    MoveL Offs(pOrigin,288.98,232.47,0.00),v40,fine,tPen\WObj:=wPaper;
    MoveL Offs(pOrigin,288.98,232.47,6.00),v60,z5,tPen\WObj:=wPaper;
    MoveL Offs(pOrigin,289.43,235.01,6.00),vTravel,z5,tPen\WObj:=wPaper;
    MoveL Offs(pOrigin,289.43,235.01,0.00),v60,z0,tPen\WObj:=wPaper;
    MoveL Offs(pOrigin,291.98,232.46,0.00),v40,fine,tPen\WObj:=wPaper;
    MoveL Offs(pOrigin,291.98,232.46,6.00),v60,z5,tPen\WObj:=wPaper;
    MoveL Offs(pOrigin,289.94,234.98,6.00),vTravel,z5,tPen\WObj:=wPaper;
    MoveL Offs(pOrigin,289.94,234.98,0.00),v60,z0,tPen\WObj:=wPaper;
    MoveL Offs(pOrigin,294.45,239.49,0.00),v40,z0,tPen\WObj:=wPaper;
    MoveL Offs(pOrigin,294.95,239.94,0.00),v40,z0,tPen\WObj:=wPaper;
    MoveL Offs(pOrigin,296.91,237.98,0.00),v40,z0,tPen\WObj:=wPaper;
    MoveL Offs(pOrigin,296.33,238.32,0.00),v40,z0,tPen\WObj:=wPaper;
    MoveL Offs(pOrigin,296.96,238.96,0.00),v40,z0,tPen\WObj:=wPaper;
    MoveL Offs(pOrigin,296.33,238.32,0.00),v40,z0,tPen\WObj:=wPaper;
    MoveL Offs(pOrigin,296.54,238.87,0.00),v40,z0,tPen\WObj:=wPaper;
    MoveL Offs(pOrigin,295.05,238.87,0.00),v40,z0,tPen\WObj:=wPaper;
    MoveL Offs(pOrigin,295.48,239.60,0.00),v40,z0,tPen\WObj:=wPaper;
    MoveL Offs(pOrigin,296.11,240.24,0.00),v40,z0,tPen\WObj:=wPaper;
    MoveL Offs(pOrigin,295.48,239.60,0.00),v40,z0,tPen\WObj:=wPaper;
    MoveL Offs(pOrigin,296.32,239.93,0.00),v40,z0,tPen\WObj:=wPaper;
    MoveL Offs(pOrigin,297.81,239.93,0.00),v40,z0,tPen\WObj:=wPaper;
    MoveL Offs(pOrigin,297.81,239.39,0.00),v40,z0,tPen\WObj:=wPaper;
    MoveL Offs(pOrigin,298.45,239.81,0.00),v40,z0,tPen\WObj:=wPaper;
    MoveL Offs(pOrigin,300.15,239.81,0.00),v40,z0,tPen\WObj:=wPaper;
    MoveL Offs(pOrigin,300.29,239.36,0.00),v40,z0,tPen\WObj:=wPaper;
    MoveL Offs(pOrigin,301.19,240.26,0.00),v40,z0,tPen\WObj:=wPaper;
    MoveL Offs(pOrigin,301.54,240.82,0.00),v40,z0,tPen\WObj:=wPaper;
    MoveL Offs(pOrigin,303.95,238.41,0.00),v40,z0,tPen\WObj:=wPaper;
    MoveL Offs(pOrigin,303.29,239.37,0.00),v40,z0,tPen\WObj:=wPaper;
    MoveL Offs(pOrigin,304.19,240.27,0.00),v40,z0,tPen\WObj:=wPaper;
    MoveL Offs(pOrigin,304.39,240.96,0.00),v40,z0,tPen\WObj:=wPaper;
    MoveL Offs(pOrigin,306.79,238.55,0.00),v40,z0,tPen\WObj:=wPaper;
    MoveL Offs(pOrigin,306.13,239.22,0.00),v40,z0,tPen\WObj:=wPaper;
    MoveL Offs(pOrigin,307.19,240.28,0.00),v40,z0,tPen\WObj:=wPaper;
    MoveL Offs(pOrigin,307.23,241.10,0.00),v40,z0,tPen\WObj:=wPaper;
    MoveL Offs(pOrigin,309.79,238.54,0.00),v40,z0,tPen\WObj:=wPaper;
  ENDPROC

  PROC DrawPart194()
    MoveL Offs(pOrigin,309.13,239.23,0.00),v40,z0,tPen\WObj:=wPaper;
    MoveL Offs(pOrigin,310.48,240.59,0.00),v40,z0,tPen\WObj:=wPaper;
    MoveL Offs(pOrigin,310.38,240.94,0.00),v40,z0,tPen\WObj:=wPaper;
    MoveL Offs(pOrigin,313.08,238.23,0.00),v40,z0,tPen\WObj:=wPaper;
    MoveL Offs(pOrigin,313.32,238.95,0.00),v40,z0,tPen\WObj:=wPaper;
    MoveL Offs(pOrigin,314.68,240.30,0.00),v40,z0,tPen\WObj:=wPaper;
    MoveL Offs(pOrigin,314.87,240.92,0.00),v40,z0,tPen\WObj:=wPaper;
    MoveL Offs(pOrigin,317.58,238.22,0.00),v40,z0,tPen\WObj:=wPaper;
    MoveL Offs(pOrigin,317.67,238.81,0.00),v40,z0,tPen\WObj:=wPaper;
    MoveL Offs(pOrigin,319.02,240.16,0.00),v40,z0,tPen\WObj:=wPaper;
    MoveL Offs(pOrigin,319.67,240.61,0.00),v40,z0,tPen\WObj:=wPaper;
    MoveL Offs(pOrigin,322.52,237.76,0.00),v40,z0,tPen\WObj:=wPaper;
    MoveL Offs(pOrigin,322.01,238.67,0.00),v40,z0,tPen\WObj:=wPaper;
    MoveL Offs(pOrigin,323.51,240.18,0.00),v40,z0,tPen\WObj:=wPaper;
    MoveL Offs(pOrigin,324.31,240.45,0.00),v40,z0,tPen\WObj:=wPaper;
    MoveL Offs(pOrigin,327.17,237.59,0.00),v40,z0,tPen\WObj:=wPaper;
    MoveL Offs(pOrigin,327.70,238.39,0.00),v40,z0,tPen\WObj:=wPaper;
    MoveL Offs(pOrigin,329.06,239.74,0.00),v40,z0,tPen\WObj:=wPaper;
    MoveL Offs(pOrigin,329.11,240.13,0.00),v40,z0,tPen\WObj:=wPaper;
    MoveL Offs(pOrigin,332.11,237.13,0.00),v40,z0,tPen\WObj:=wPaper;
    MoveL Offs(pOrigin,331.75,237.95,0.00),v40,z0,tPen\WObj:=wPaper;
    MoveL Offs(pOrigin,333.10,239.31,0.00),v40,z0,tPen\WObj:=wPaper;
    MoveL Offs(pOrigin,333.90,239.82,0.00),v40,z0,tPen\WObj:=wPaper;
    MoveL Offs(pOrigin,337.06,236.66,0.00),v40,z0,tPen\WObj:=wPaper;
    MoveL Offs(pOrigin,337.29,237.52,0.00),v40,z0,tPen\WObj:=wPaper;
    MoveL Offs(pOrigin,338.49,238.72,0.00),v40,z0,tPen\WObj:=wPaper;
    MoveL Offs(pOrigin,339.15,239.05,0.00),v40,z0,tPen\WObj:=wPaper;
    MoveL Offs(pOrigin,341.85,236.35,0.00),v40,z0,tPen\WObj:=wPaper;
    MoveL Offs(pOrigin,342.53,236.79,0.00),v40,z0,tPen\WObj:=wPaper;
    MoveL Offs(pOrigin,343.88,238.14,0.00),v40,z0,tPen\WObj:=wPaper;
    MoveL Offs(pOrigin,344.09,238.59,0.00),v40,z0,tPen\WObj:=wPaper;
    MoveL Offs(pOrigin,347.10,235.58,0.00),v40,z0,tPen\WObj:=wPaper;
    MoveL Offs(pOrigin,346.72,236.50,0.00),v40,z0,tPen\WObj:=wPaper;
    MoveL Offs(pOrigin,347.92,237.70,0.00),v40,z0,tPen\WObj:=wPaper;
    MoveL Offs(pOrigin,347.39,238.28,0.00),v40,z0,tPen\WObj:=wPaper;
    MoveL Offs(pOrigin,350.54,235.12,0.00),v40,z0,tPen\WObj:=wPaper;
    MoveL Offs(pOrigin,350.76,236.07,0.00),v40,z0,tPen\WObj:=wPaper;
    MoveL Offs(pOrigin,351.82,237.12,0.00),v40,z0,tPen\WObj:=wPaper;
    MoveL Offs(pOrigin,352.78,237.36,0.00),v40,z0,tPen\WObj:=wPaper;
    MoveL Offs(pOrigin,355.64,234.51,0.00),v40,z0,tPen\WObj:=wPaper;
    MoveL Offs(pOrigin,356.01,235.33,0.00),v40,z0,tPen\WObj:=wPaper;
    MoveL Offs(pOrigin,357.06,236.38,0.00),v40,fine,tPen\WObj:=wPaper;
    MoveL Offs(pOrigin,357.06,236.38,6.00),v60,z5,tPen\WObj:=wPaper;
    MoveL Offs(pOrigin,357.59,234.05,6.00),vTravel,z5,tPen\WObj:=wPaper;
    MoveL Offs(pOrigin,357.59,234.05,0.00),v60,z0,tPen\WObj:=wPaper;
    MoveL Offs(pOrigin,354.43,237.21,0.00),v40,fine,tPen\WObj:=wPaper;
    MoveL Offs(pOrigin,354.43,237.21,6.00),v60,z5,tPen\WObj:=wPaper;
    MoveL Offs(pOrigin,353.16,236.97,6.00),vTravel,z5,tPen\WObj:=wPaper;
    MoveL Offs(pOrigin,353.16,236.97,0.00),v60,z0,tPen\WObj:=wPaper;
    MoveL Offs(pOrigin,352.11,235.92,0.00),v40,z0,tPen\WObj:=wPaper;
    MoveL Offs(pOrigin,352.19,234.97,0.00),v40,z0,tPen\WObj:=wPaper;
    MoveL Offs(pOrigin,349.19,237.97,0.00),v40,z0,tPen\WObj:=wPaper;
    MoveL Offs(pOrigin,349.27,237.56,0.00),v40,z0,tPen\WObj:=wPaper;
    MoveL Offs(pOrigin,348.22,236.51,0.00),v40,fine,tPen\WObj:=wPaper;
    MoveL Offs(pOrigin,348.22,236.51,6.00),v60,z5,tPen\WObj:=wPaper;
    MoveL Offs(pOrigin,346.73,238.00,6.00),vTravel,z5,tPen\WObj:=wPaper;
    MoveL Offs(pOrigin,346.73,238.00,0.00),v60,z0,tPen\WObj:=wPaper;
    MoveL Offs(pOrigin,345.37,236.65,0.00),v40,z0,tPen\WObj:=wPaper;
    MoveL Offs(pOrigin,345.30,235.89,0.00),v40,z0,tPen\WObj:=wPaper;
    MoveL Offs(pOrigin,342.29,238.89,0.00),v40,z0,tPen\WObj:=wPaper;
    MoveL Offs(pOrigin,342.68,238.44,0.00),v40,z0,tPen\WObj:=wPaper;
    MoveL Offs(pOrigin,341.33,237.09,0.00),v40,fine,tPen\WObj:=wPaper;
    MoveL Offs(pOrigin,341.33,237.09,6.00),v60,z5,tPen\WObj:=wPaper;
    MoveL Offs(pOrigin,339.84,238.58,6.00),vTravel,z5,tPen\WObj:=wPaper;
    MoveL Offs(pOrigin,339.84,238.58,0.00),v60,z0,tPen\WObj:=wPaper;
    MoveL Offs(pOrigin,338.79,237.53,0.00),v40,z0,tPen\WObj:=wPaper;
    MoveL Offs(pOrigin,338.55,236.66,0.00),v40,z0,tPen\WObj:=wPaper;
    MoveL Offs(pOrigin,335.70,239.51,0.00),v40,z0,tPen\WObj:=wPaper;
    MoveL Offs(pOrigin,335.79,239.02,0.00),v40,z0,tPen\WObj:=wPaper;
    MoveL Offs(pOrigin,334.44,237.66,0.00),v40,z0,tPen\WObj:=wPaper;
    MoveL Offs(pOrigin,333.61,237.12,0.00),v40,z0,tPen\WObj:=wPaper;
    MoveL Offs(pOrigin,330.75,239.98,0.00),v40,z0,tPen\WObj:=wPaper;
    MoveL Offs(pOrigin,330.40,239.60,0.00),v40,z0,tPen\WObj:=wPaper;
    MoveL Offs(pOrigin,329.05,238.25,0.00),v40,z0,tPen\WObj:=wPaper;
    MoveL Offs(pOrigin,328.66,237.59,0.00),v40,z0,tPen\WObj:=wPaper;
    MoveL Offs(pOrigin,325.81,240.44,0.00),v40,z0,tPen\WObj:=wPaper;
    MoveL Offs(pOrigin,326.36,240.04,0.00),v40,z0,tPen\WObj:=wPaper;
    MoveL Offs(pOrigin,325.01,238.68,0.00),v40,fine,tPen\WObj:=wPaper;
    MoveL Offs(pOrigin,325.01,238.68,6.00),v60,z5,tPen\WObj:=wPaper;
    MoveL Offs(pOrigin,324.86,240.03,6.00),vTravel,z5,tPen\WObj:=wPaper;
    MoveL Offs(pOrigin,324.86,240.03,0.00),v60,z0,tPen\WObj:=wPaper;
    MoveL Offs(pOrigin,323.51,238.68,0.00),v40,z0,tPen\WObj:=wPaper;
    MoveL Offs(pOrigin,324.02,237.75,0.00),v40,z0,tPen\WObj:=wPaper;
    MoveL Offs(pOrigin,321.17,240.61,0.00),v40,z0,tPen\WObj:=wPaper;
    MoveL Offs(pOrigin,320.52,240.17,0.00),v40,z0,tPen\WObj:=wPaper;
    MoveL Offs(pOrigin,319.17,238.81,0.00),v40,z0,tPen\WObj:=wPaper;
    MoveL Offs(pOrigin,319.23,238.07,0.00),v40,z0,tPen\WObj:=wPaper;
    MoveL Offs(pOrigin,316.37,240.92,0.00),v40,z0,tPen\WObj:=wPaper;
    MoveL Offs(pOrigin,316.17,240.30,0.00),v40,z0,tPen\WObj:=wPaper;
    MoveL Offs(pOrigin,314.82,238.95,0.00),v40,z0,tPen\WObj:=wPaper;
    MoveL Offs(pOrigin,314.58,238.23,0.00),v40,z0,tPen\WObj:=wPaper;
    MoveL Offs(pOrigin,311.88,240.93,0.00),v40,z0,tPen\WObj:=wPaper;
    MoveL Offs(pOrigin,311.98,240.59,0.00),v40,z0,tPen\WObj:=wPaper;
    MoveL Offs(pOrigin,310.63,239.24,0.00),v40,fine,tPen\WObj:=wPaper;
    MoveL Offs(pOrigin,310.63,239.24,6.00),v60,z5,tPen\WObj:=wPaper;
    MoveL Offs(pOrigin,300.80,238.57,6.00),vTravel,z5,tPen\WObj:=wPaper;
    MoveL Offs(pOrigin,300.80,238.57,0.00),v60,z0,tPen\WObj:=wPaper;
    MoveL Offs(pOrigin,296.44,242.93,0.00),v40,fine,tPen\WObj:=wPaper;
    MoveL Offs(pOrigin,296.44,242.93,6.00),v60,z5,tPen\WObj:=wPaper;
    MoveL Offs(pOrigin,296.96,240.98,6.00),vTravel,z5,tPen\WObj:=wPaper;
    MoveL Offs(pOrigin,296.96,240.98,0.00),v60,z0,tPen\WObj:=wPaper;
    MoveL Offs(pOrigin,298.02,240.98,0.00),v40,z0,tPen\WObj:=wPaper;
    MoveL Offs(pOrigin,298.65,240.70,0.00),v40,z0,tPen\WObj:=wPaper;
    MoveL Offs(pOrigin,295.64,237.69,0.00),v40,z0,tPen\WObj:=wPaper;
    MoveL Offs(pOrigin,296.01,237.39,0.00),v40,z0,tPen\WObj:=wPaper;
    MoveL Offs(pOrigin,293.60,239.79,0.00),v40,z0,tPen\WObj:=wPaper;
    MoveL Offs(pOrigin,292.92,238.87,0.00),v40,z0,tPen\WObj:=wPaper;
    MoveL Offs(pOrigin,291.01,238.87,0.00),v40,z0,tPen\WObj:=wPaper;
    MoveL Offs(pOrigin,291.01,237.82,0.00),v40,z0,tPen\WObj:=wPaper;
    MoveL Offs(pOrigin,294.41,237.82,0.00),v40,z0,tPen\WObj:=wPaper;
    MoveL Offs(pOrigin,294.96,236.94,0.00),v40,z0,tPen\WObj:=wPaper;
    MoveL Offs(pOrigin,290.00,241.90,0.00),v40,z0,tPen\WObj:=wPaper;
    MoveL Offs(pOrigin,290.56,241.57,0.00),v40,z0,tPen\WObj:=wPaper;
    MoveL Offs(pOrigin,291.61,242.62,0.00),v40,z0,tPen\WObj:=wPaper;
    MoveL Offs(pOrigin,292.40,242.49,0.00),v40,z0,tPen\WObj:=wPaper;
    MoveL Offs(pOrigin,289.99,244.90,0.00),v40,fine,tPen\WObj:=wPaper;
    MoveL Offs(pOrigin,289.99,244.90,6.00),v60,z5,tPen\WObj:=wPaper;
    MoveL Offs(pOrigin,289.99,246.39,6.00),vTravel,z5,tPen\WObj:=wPaper;
    MoveL Offs(pOrigin,289.99,246.39,0.00),v60,z0,tPen\WObj:=wPaper;
    MoveL Offs(pOrigin,291.94,244.44,0.00),v40,fine,tPen\WObj:=wPaper;
  ENDPROC

  PROC DrawPart195()
    MoveL Offs(pOrigin,291.94,244.44,6.00),v60,z5,tPen\WObj:=wPaper;
    MoveL Offs(pOrigin,291.94,245.94,6.00),vTravel,z5,tPen\WObj:=wPaper;
    MoveL Offs(pOrigin,291.94,245.94,0.00),v60,z0,tPen\WObj:=wPaper;
    MoveL Offs(pOrigin,289.98,247.89,0.00),v40,fine,tPen\WObj:=wPaper;
    MoveL Offs(pOrigin,289.98,247.89,6.00),v60,z5,tPen\WObj:=wPaper;
    MoveL Offs(pOrigin,291.65,250.44,6.00),vTravel,z5,tPen\WObj:=wPaper;
    MoveL Offs(pOrigin,291.65,250.44,0.00),v60,z0,tPen\WObj:=wPaper;
    MoveL Offs(pOrigin,292.71,251.71,0.00),v40,z0,tPen\WObj:=wPaper;
    MoveL Offs(pOrigin,291.65,250.44,0.00),v40,fine,tPen\WObj:=wPaper;
    MoveL Offs(pOrigin,291.65,250.44,6.00),v60,z5,tPen\WObj:=wPaper;
    MoveL Offs(pOrigin,297.18,246.67,6.00),vTravel,z5,tPen\WObj:=wPaper;
    MoveL Offs(pOrigin,297.18,246.67,0.00),v60,z0,tPen\WObj:=wPaper;
    MoveL Offs(pOrigin,300.03,243.82,0.00),v40,z0,tPen\WObj:=wPaper;
    MoveL Offs(pOrigin,299.44,242.92,0.00),v40,z0,tPen\WObj:=wPaper;
    MoveL Offs(pOrigin,296.73,245.62,0.00),v40,z0,tPen\WObj:=wPaper;
    MoveL Offs(pOrigin,297.31,245.34,0.00),v40,z0,tPen\WObj:=wPaper;
    MoveL Offs(pOrigin,300.02,248.04,0.00),v40,fine,tPen\WObj:=wPaper;
    MoveL Offs(pOrigin,300.02,248.04,6.00),v60,z5,tPen\WObj:=wPaper;
    MoveL Offs(pOrigin,300.36,246.26,6.00),vTravel,z5,tPen\WObj:=wPaper;
    MoveL Offs(pOrigin,300.36,246.26,0.00),v60,z0,tPen\WObj:=wPaper;
    MoveL Offs(pOrigin,298.24,246.26,0.00),v40,z0,tPen\WObj:=wPaper;
    MoveL Offs(pOrigin,298.86,246.40,0.00),v40,z0,tPen\WObj:=wPaper;
    MoveL Offs(pOrigin,298.86,245.34,0.00),v40,z0,tPen\WObj:=wPaper;
    MoveL Offs(pOrigin,298.02,245.21,0.00),v40,z0,tPen\WObj:=wPaper;
    MoveL Offs(pOrigin,333.94,245.21,0.00),v40,fine,tPen\WObj:=wPaper;
    MoveL Offs(pOrigin,333.94,245.21,6.00),v60,z5,tPen\WObj:=wPaper;
    MoveL Offs(pOrigin,335.21,244.15,6.00),vTravel,z5,tPen\WObj:=wPaper;
    MoveL Offs(pOrigin,335.21,244.15,0.00),v60,z0,tPen\WObj:=wPaper;
    MoveL Offs(pOrigin,347.33,244.15,0.00),v40,z0,tPen\WObj:=wPaper;
    MoveL Offs(pOrigin,347.54,243.10,0.00),v40,z0,tPen\WObj:=wPaper;
    MoveL Offs(pOrigin,356.46,243.10,0.00),v40,fine,tPen\WObj:=wPaper;
    MoveL Offs(pOrigin,356.46,243.10,6.00),v60,z5,tPen\WObj:=wPaper;
    MoveL Offs(pOrigin,354.08,243.87,6.00),vTravel,z5,tPen\WObj:=wPaper;
    MoveL Offs(pOrigin,354.08,243.87,0.00),v60,z0,tPen\WObj:=wPaper;
    MoveL Offs(pOrigin,352.43,242.21,0.00),v40,fine,tPen\WObj:=wPaper;
    MoveL Offs(pOrigin,352.43,242.21,6.00),v60,z5,tPen\WObj:=wPaper;
    MoveL Offs(pOrigin,348.84,244.60,6.00),vTravel,z5,tPen\WObj:=wPaper;
    MoveL Offs(pOrigin,348.84,244.60,0.00),v60,z0,tPen\WObj:=wPaper;
    MoveL Offs(pOrigin,347.04,242.79,0.00),v40,fine,tPen\WObj:=wPaper;
    MoveL Offs(pOrigin,347.04,242.79,6.00),v60,z5,tPen\WObj:=wPaper;
    MoveL Offs(pOrigin,339.26,245.47,6.00),vTravel,z5,tPen\WObj:=wPaper;
    MoveL Offs(pOrigin,339.26,245.47,0.00),v60,z0,tPen\WObj:=wPaper;
    MoveL Offs(pOrigin,337.61,243.81,0.00),v40,fine,tPen\WObj:=wPaper;
    MoveL Offs(pOrigin,337.61,243.81,6.00),v60,z5,tPen\WObj:=wPaper;
    MoveL Offs(pOrigin,334.45,239.16,6.00),vTravel,z5,tPen\WObj:=wPaper;
    MoveL Offs(pOrigin,334.45,239.16,0.00),v60,z0,tPen\WObj:=wPaper;
    MoveL Offs(pOrigin,333.09,237.81,0.00),v40,fine,tPen\WObj:=wPaper;
    MoveL Offs(pOrigin,333.09,237.81,6.00),v60,z5,tPen\WObj:=wPaper;
    MoveL Offs(pOrigin,328.65,243.58,6.00),vTravel,z5,tPen\WObj:=wPaper;
    MoveL Offs(pOrigin,328.65,243.58,0.00),v60,z0,tPen\WObj:=wPaper;
    MoveL Offs(pOrigin,325.49,246.73,0.00),v40,fine,tPen\WObj:=wPaper;
    MoveL Offs(pOrigin,325.49,246.73,6.00),v60,z5,tPen\WObj:=wPaper;
    MoveL Offs(pOrigin,329.22,244.39,6.00),vTravel,z5,tPen\WObj:=wPaper;
    MoveL Offs(pOrigin,329.22,244.39,0.00),v60,z0,tPen\WObj:=wPaper;
    MoveL Offs(pOrigin,331.02,246.19,0.00),v40,fine,tPen\WObj:=wPaper;
    MoveL Offs(pOrigin,331.02,246.19,6.00),v60,z5,tPen\WObj:=wPaper;
    MoveL Offs(pOrigin,357.52,239.60,6.00),vTravel,z5,tPen\WObj:=wPaper;
    MoveL Offs(pOrigin,357.52,239.60,0.00),v60,z0,tPen\WObj:=wPaper;
    MoveL Offs(pOrigin,364.75,239.39,0.00),v40,z0,tPen\WObj:=wPaper;
    MoveL Offs(pOrigin,369.21,237.97,0.00),v40,z0,tPen\WObj:=wPaper;
    MoveL Offs(pOrigin,371.55,236.62,0.00),v40,z0,tPen\WObj:=wPaper;
    MoveL Offs(pOrigin,373.25,235.14,0.00),v40,z0,tPen\WObj:=wPaper;
    MoveL Offs(pOrigin,374.81,233.01,0.00),v40,z0,tPen\WObj:=wPaper;
    MoveL Offs(pOrigin,375.87,230.68,0.00),v40,z0,tPen\WObj:=wPaper;
    MoveL Offs(pOrigin,377.08,226.64,0.00),v40,z0,tPen\WObj:=wPaper;
    MoveL Offs(pOrigin,377.71,221.96,0.00),v40,z0,tPen\WObj:=wPaper;
    MoveL Offs(pOrigin,377.71,212.82,0.00),v40,z0,tPen\WObj:=wPaper;
    MoveL Offs(pOrigin,376.86,204.96,0.00),v40,z0,tPen\WObj:=wPaper;
    MoveL Offs(pOrigin,373.89,190.51,0.00),v40,z0,tPen\WObj:=wPaper;
    MoveL Offs(pOrigin,376.23,188.60,0.00),v40,z0,tPen\WObj:=wPaper;
    MoveL Offs(pOrigin,377.92,186.48,0.00),v40,z0,tPen\WObj:=wPaper;
    MoveL Offs(pOrigin,378.14,186.07,0.00),v40,z0,tPen\WObj:=wPaper;
    MoveL Offs(pOrigin,375.80,186.07,0.00),v40,z0,tPen\WObj:=wPaper;
    MoveL Offs(pOrigin,375.80,185.02,0.00),v40,z0,tPen\WObj:=wPaper;
    MoveL Offs(pOrigin,378.35,185.02,0.00),v40,z0,tPen\WObj:=wPaper;
    MoveL Offs(pOrigin,378.77,185.62,0.00),v40,z0,tPen\WObj:=wPaper;
    MoveL Offs(pOrigin,378.99,186.90,0.00),v40,z0,tPen\WObj:=wPaper;
    MoveL Offs(pOrigin,378.99,186.90,0.00),v40,z0,tPen\WObj:=wPaper;
    MoveL Offs(pOrigin,381.11,199.86,0.00),v40,z0,tPen\WObj:=wPaper;
    MoveL Offs(pOrigin,381.96,211.12,0.00),v40,z0,tPen\WObj:=wPaper;
    MoveL Offs(pOrigin,381.54,221.96,0.00),v40,z0,tPen\WObj:=wPaper;
    MoveL Offs(pOrigin,381.11,224.94,0.00),v40,z0,tPen\WObj:=wPaper;
    MoveL Offs(pOrigin,379.41,230.68,0.00),v40,z0,tPen\WObj:=wPaper;
    MoveL Offs(pOrigin,379.41,231.52,0.00),v40,z0,tPen\WObj:=wPaper;
    MoveL Offs(pOrigin,379.84,231.48,0.00),v40,z0,tPen\WObj:=wPaper;
    MoveL Offs(pOrigin,381.54,231.48,0.00),v40,z0,tPen\WObj:=wPaper;
    MoveL Offs(pOrigin,381.75,231.52,0.00),v40,z0,tPen\WObj:=wPaper;
    MoveL Offs(pOrigin,381.54,231.95,0.00),v40,z0,tPen\WObj:=wPaper;
    MoveL Offs(pOrigin,381.75,231.52,0.00),v40,z0,tPen\WObj:=wPaper;
    MoveL Offs(pOrigin,381.91,231.37,0.00),v40,z0,tPen\WObj:=wPaper;
    MoveL Offs(pOrigin,378.90,228.36,0.00),v40,z0,tPen\WObj:=wPaper;
    MoveL Offs(pOrigin,378.46,229.41,0.00),v40,z0,tPen\WObj:=wPaper;
    MoveL Offs(pOrigin,381.46,232.41,0.00),v40,fine,tPen\WObj:=wPaper;
    MoveL Offs(pOrigin,381.46,232.41,6.00),v60,z5,tPen\WObj:=wPaper;
    MoveL Offs(pOrigin,382.61,231.43,6.00),vTravel,z5,tPen\WObj:=wPaper;
    MoveL Offs(pOrigin,382.61,231.43,0.00),v60,z0,tPen\WObj:=wPaper;
    MoveL Offs(pOrigin,374.50,239.54,0.00),v40,z0,tPen\WObj:=wPaper;
    MoveL Offs(pOrigin,374.59,238.98,0.00),v40,z0,tPen\WObj:=wPaper;
    MoveL Offs(pOrigin,373.24,237.63,0.00),v40,z0,tPen\WObj:=wPaper;
    MoveL Offs(pOrigin,373.89,237.48,0.00),v40,z0,tPen\WObj:=wPaper;
    MoveL Offs(pOrigin,374.10,237.05,0.00),v40,z0,tPen\WObj:=wPaper;
    MoveL Offs(pOrigin,373.89,237.48,0.00),v40,fine,tPen\WObj:=wPaper;
    MoveL Offs(pOrigin,373.89,237.48,6.00),v60,z5,tPen\WObj:=wPaper;
    MoveL Offs(pOrigin,373.67,238.87,6.00),vTravel,z5,tPen\WObj:=wPaper;
    MoveL Offs(pOrigin,373.67,238.87,0.00),v60,z0,tPen\WObj:=wPaper;
    MoveL Offs(pOrigin,371.12,238.87,0.00),v40,fine,tPen\WObj:=wPaper;
    MoveL Offs(pOrigin,371.12,238.87,6.00),v60,z5,tPen\WObj:=wPaper;
    MoveL Offs(pOrigin,371.65,240.90,6.00),vTravel,z5,tPen\WObj:=wPaper;
    MoveL Offs(pOrigin,371.65,240.90,0.00),v60,z0,tPen\WObj:=wPaper;
    MoveL Offs(pOrigin,383.67,228.88,0.00),v40,z0,tPen\WObj:=wPaper;
    MoveL Offs(pOrigin,383.40,228.38,0.00),v40,z0,tPen\WObj:=wPaper;
    MoveL Offs(pOrigin,381.89,226.87,0.00),v40,z0,tPen\WObj:=wPaper;
    MoveL Offs(pOrigin,381.14,226.12,0.00),v40,z0,tPen\WObj:=wPaper;
    MoveL Offs(pOrigin,379.49,224.47,0.00),v40,z0,tPen\WObj:=wPaper;
    MoveL Offs(pOrigin,378.89,224.70,0.00),v40,z0,tPen\WObj:=wPaper;
    MoveL Offs(pOrigin,386.40,217.19,0.00),v40,z0,tPen\WObj:=wPaper;
    MoveL Offs(pOrigin,385.91,217.45,0.00),v40,z0,tPen\WObj:=wPaper;
    MoveL Offs(pOrigin,384.26,215.80,0.00),v40,z0,tPen\WObj:=wPaper;
    MoveL Offs(pOrigin,383.56,215.55,0.00),v40,z0,tPen\WObj:=wPaper;
    MoveL Offs(pOrigin,387.01,212.09,0.00),v40,z0,tPen\WObj:=wPaper;
  ENDPROC

  PROC DrawPart196()
    MoveL Offs(pOrigin,386.64,212.21,0.00),v40,z0,tPen\WObj:=wPaper;
    MoveL Offs(pOrigin,384.84,210.40,0.00),v40,z0,tPen\WObj:=wPaper;
    MoveL Offs(pOrigin,384.32,210.30,0.00),v40,z0,tPen\WObj:=wPaper;
    MoveL Offs(pOrigin,387.48,207.15,0.00),v40,z0,tPen\WObj:=wPaper;
    MoveL Offs(pOrigin,386.93,206.52,0.00),v40,z0,tPen\WObj:=wPaper;
    MoveL Offs(pOrigin,385.27,204.86,0.00),v40,z0,tPen\WObj:=wPaper;
    MoveL Offs(pOrigin,384.49,205.66,0.00),v40,z0,tPen\WObj:=wPaper;
    MoveL Offs(pOrigin,387.79,202.35,0.00),v40,z0,tPen\WObj:=wPaper;
    MoveL Offs(pOrigin,387.36,202.47,0.00),v40,z0,tPen\WObj:=wPaper;
    MoveL Offs(pOrigin,385.56,200.67,0.00),v40,z0,tPen\WObj:=wPaper;
    MoveL Offs(pOrigin,384.95,200.71,0.00),v40,z0,tPen\WObj:=wPaper;
    MoveL Offs(pOrigin,388.26,197.41,0.00),v40,z0,tPen\WObj:=wPaper;
    MoveL Offs(pOrigin,387.79,196.93,0.00),v40,z0,tPen\WObj:=wPaper;
    MoveL Offs(pOrigin,385.99,195.13,0.00),v40,z0,tPen\WObj:=wPaper;
    MoveL Offs(pOrigin,385.42,195.77,0.00),v40,z0,tPen\WObj:=wPaper;
    MoveL Offs(pOrigin,388.72,192.46,0.00),v40,z0,tPen\WObj:=wPaper;
    MoveL Offs(pOrigin,388.38,193.04,0.00),v40,z0,tPen\WObj:=wPaper;
    MoveL Offs(pOrigin,386.43,191.09,0.00),v40,z0,tPen\WObj:=wPaper;
    MoveL Offs(pOrigin,385.88,190.82,0.00),v40,z0,tPen\WObj:=wPaper;
    MoveL Offs(pOrigin,389.19,187.52,0.00),v40,z0,tPen\WObj:=wPaper;
    MoveL Offs(pOrigin,388.81,187.50,0.00),v40,z0,tPen\WObj:=wPaper;
    MoveL Offs(pOrigin,387.01,185.69,0.00),v40,z0,tPen\WObj:=wPaper;
    MoveL Offs(pOrigin,386.35,185.88,0.00),v40,z0,tPen\WObj:=wPaper;
    MoveL Offs(pOrigin,389.80,182.42,0.00),v40,z0,tPen\WObj:=wPaper;
    MoveL Offs(pOrigin,389.25,181.96,0.00),v40,z0,tPen\WObj:=wPaper;
    MoveL Offs(pOrigin,387.44,180.15,0.00),v40,z0,tPen\WObj:=wPaper;
    MoveL Offs(pOrigin,386.97,179.29,0.00),v40,z0,tPen\WObj:=wPaper;
    MoveL Offs(pOrigin,390.42,175.83,0.00),v40,z0,tPen\WObj:=wPaper;
    MoveL Offs(pOrigin,389.83,176.57,0.00),v40,z0,tPen\WObj:=wPaper;
    MoveL Offs(pOrigin,387.88,174.61,0.00),v40,z0,tPen\WObj:=wPaper;
    MoveL Offs(pOrigin,387.43,174.34,0.00),v40,z0,tPen\WObj:=wPaper;
    MoveL Offs(pOrigin,390.89,170.88,0.00),v40,z0,tPen\WObj:=wPaper;
    MoveL Offs(pOrigin,390.26,171.02,0.00),v40,z0,tPen\WObj:=wPaper;
    MoveL Offs(pOrigin,388.46,169.22,0.00),v40,z0,tPen\WObj:=wPaper;
    MoveL Offs(pOrigin,388.98,169.18,0.00),v40,z0,tPen\WObj:=wPaper;
    MoveL Offs(pOrigin,390.04,169.18,0.00),v40,z0,tPen\WObj:=wPaper;
    MoveL Offs(pOrigin,390.41,169.68,0.00),v40,z0,tPen\WObj:=wPaper;
    MoveL Offs(pOrigin,388.45,167.72,0.00),v40,z0,tPen\WObj:=wPaper;
    MoveL Offs(pOrigin,388.05,167.75,0.00),v40,z0,tPen\WObj:=wPaper;
    MoveL Offs(pOrigin,391.51,164.29,0.00),v40,z0,tPen\WObj:=wPaper;
    MoveL Offs(pOrigin,390.84,164.13,0.00),v40,z0,tPen\WObj:=wPaper;
    MoveL Offs(pOrigin,389.04,162.33,0.00),v40,z0,tPen\WObj:=wPaper;
    MoveL Offs(pOrigin,388.51,162.80,0.00),v40,z0,tPen\WObj:=wPaper;
    MoveL Offs(pOrigin,391.97,159.35,0.00),v40,z0,tPen\WObj:=wPaper;
    MoveL Offs(pOrigin,391.42,158.74,0.00),v40,z0,tPen\WObj:=wPaper;
    MoveL Offs(pOrigin,389.47,156.79,0.00),v40,z0,tPen\WObj:=wPaper;
    MoveL Offs(pOrigin,389.13,156.21,0.00),v40,z0,tPen\WObj:=wPaper;
    MoveL Offs(pOrigin,392.59,152.75,0.00),v40,z0,tPen\WObj:=wPaper;
    MoveL Offs(pOrigin,392.00,151.85,0.00),v40,z0,tPen\WObj:=wPaper;
    MoveL Offs(pOrigin,390.35,150.20,0.00),v40,z0,tPen\WObj:=wPaper;
    MoveL Offs(pOrigin,389.60,149.77,0.00),v40,z0,tPen\WObj:=wPaper;
    MoveL Offs(pOrigin,393.06,146.31,0.00),v40,z0,tPen\WObj:=wPaper;
    MoveL Offs(pOrigin,392.58,146.46,0.00),v40,z0,tPen\WObj:=wPaper;
    MoveL Offs(pOrigin,390.78,144.66,0.00),v40,z0,tPen\WObj:=wPaper;
    MoveL Offs(pOrigin,391.31,144.89,0.00),v40,z0,tPen\WObj:=wPaper;
    MoveL Offs(pOrigin,392.38,144.89,0.00),v40,z0,tPen\WObj:=wPaper;
    MoveL Offs(pOrigin,392.88,145.27,0.00),v40,z0,tPen\WObj:=wPaper;
    MoveL Offs(pOrigin,391.08,143.46,0.00),v40,z0,tPen\WObj:=wPaper;
    MoveL Offs(pOrigin,391.52,142.78,0.00),v40,z0,tPen\WObj:=wPaper;
    MoveL Offs(pOrigin,392.59,142.78,0.00),v40,fine,tPen\WObj:=wPaper;
    MoveL Offs(pOrigin,392.59,142.78,6.00),v60,z5,tPen\WObj:=wPaper;
    MoveL Offs(pOrigin,393.03,143.92,6.00),vTravel,z5,tPen\WObj:=wPaper;
    MoveL Offs(pOrigin,393.03,143.92,0.00),v60,z0,tPen\WObj:=wPaper;
    MoveL Offs(pOrigin,391.07,141.97,0.00),v40,fine,tPen\WObj:=wPaper;
    MoveL Offs(pOrigin,391.07,141.97,6.00),v60,z5,tPen\WObj:=wPaper;
    MoveL Offs(pOrigin,390.37,143.02,6.00),vTravel,z5,tPen\WObj:=wPaper;
    MoveL Offs(pOrigin,390.37,143.02,0.00),v60,z0,tPen\WObj:=wPaper;
    MoveL Offs(pOrigin,393.98,139.42,0.00),v40,fine,tPen\WObj:=wPaper;
    MoveL Offs(pOrigin,393.98,139.42,6.00),v60,z5,tPen\WObj:=wPaper;
    MoveL Offs(pOrigin,393.01,138.55,6.00),vTravel,z5,tPen\WObj:=wPaper;
    MoveL Offs(pOrigin,393.01,138.55,0.00),v60,z0,tPen\WObj:=wPaper;
    MoveL Offs(pOrigin,391.95,138.55,0.00),v40,z0,tPen\WObj:=wPaper;
    MoveL Offs(pOrigin,391.95,137.50,0.00),v40,z0,tPen\WObj:=wPaper;
    MoveL Offs(pOrigin,393.22,137.50,0.00),v40,z0,tPen\WObj:=wPaper;
    MoveL Offs(pOrigin,393.60,137.03,0.00),v40,z0,tPen\WObj:=wPaper;
    MoveL Offs(pOrigin,388.95,132.37,0.00),v40,z0,tPen\WObj:=wPaper;
    MoveL Offs(pOrigin,389.40,132.22,0.00),v40,z0,tPen\WObj:=wPaper;
    MoveL Offs(pOrigin,390.67,132.22,0.00),v40,z0,tPen\WObj:=wPaper;
    MoveL Offs(pOrigin,390.67,133.27,0.00),v40,z0,tPen\WObj:=wPaper;
    MoveL Offs(pOrigin,389.40,133.27,0.00),v40,fine,tPen\WObj:=wPaper;
    MoveL Offs(pOrigin,389.40,133.27,6.00),v60,z5,tPen\WObj:=wPaper;
    MoveL Offs(pOrigin,388.16,133.29,6.00),vTravel,z5,tPen\WObj:=wPaper;
    MoveL Offs(pOrigin,388.16,133.29,0.00),v60,z0,tPen\WObj:=wPaper;
    MoveL Offs(pOrigin,397.62,123.83,0.00),v40,z0,tPen\WObj:=wPaper;
    MoveL Offs(pOrigin,397.16,124.16,0.00),v40,z0,tPen\WObj:=wPaper;
    MoveL Offs(pOrigin,394.75,121.75,0.00),v40,z0,tPen\WObj:=wPaper;
    MoveL Offs(pOrigin,395.35,121.66,0.00),v40,z0,tPen\WObj:=wPaper;
    MoveL Offs(pOrigin,396.62,121.66,0.00),v40,z0,tPen\WObj:=wPaper;
    MoveL Offs(pOrigin,397.00,122.51,0.00),v40,z0,tPen\WObj:=wPaper;
    MoveL Offs(pOrigin,394.60,120.11,0.00),v40,z0,tPen\WObj:=wPaper;
    MoveL Offs(pOrigin,394.19,119.79,0.00),v40,z0,tPen\WObj:=wPaper;
    MoveL Offs(pOrigin,400.80,113.18,0.00),v40,fine,tPen\WObj:=wPaper;
    MoveL Offs(pOrigin,400.80,113.18,6.00),v60,z5,tPen\WObj:=wPaper;
    MoveL Offs(pOrigin,401.86,110.63,6.00),vTravel,z5,tPen\WObj:=wPaper;
    MoveL Offs(pOrigin,401.86,110.63,0.00),v60,z0,tPen\WObj:=wPaper;
    MoveL Offs(pOrigin,394.19,118.30,0.00),v40,fine,tPen\WObj:=wPaper;
    MoveL Offs(pOrigin,394.19,118.30,6.00),v60,z5,tPen\WObj:=wPaper;
    MoveL Offs(pOrigin,395.35,119.54,6.00),vTravel,z5,tPen\WObj:=wPaper;
    MoveL Offs(pOrigin,395.35,119.54,0.00),v60,z0,tPen\WObj:=wPaper;
    MoveL Offs(pOrigin,396.62,119.54,0.00),v40,z0,tPen\WObj:=wPaper;
    MoveL Offs(pOrigin,396.41,120.60,0.00),v40,z0,tPen\WObj:=wPaper;
    MoveL Offs(pOrigin,395.35,120.60,0.00),v40,fine,tPen\WObj:=wPaper;
    MoveL Offs(pOrigin,395.35,120.60,6.00),v60,z5,tPen\WObj:=wPaper;
    MoveL Offs(pOrigin,394.18,121.29,6.00),vTravel,z5,tPen\WObj:=wPaper;
    MoveL Offs(pOrigin,394.18,121.29,0.00),v60,z0,tPen\WObj:=wPaper;
    MoveL Offs(pOrigin,398.54,116.93,0.00),v40,fine,tPen\WObj:=wPaper;
    MoveL Offs(pOrigin,398.54,116.93,6.00),v60,z5,tPen\WObj:=wPaper;
    MoveL Offs(pOrigin,397.81,111.69,6.00),vTravel,z5,tPen\WObj:=wPaper;
    MoveL Offs(pOrigin,397.81,111.69,0.00),v60,z0,tPen\WObj:=wPaper;
    MoveL Offs(pOrigin,402.92,106.58,0.00),v40,fine,tPen\WObj:=wPaper;
    MoveL Offs(pOrigin,402.92,106.58,6.00),v60,z5,tPen\WObj:=wPaper;
    MoveL Offs(pOrigin,403.21,104.24,6.00),vTravel,z5,tPen\WObj:=wPaper;
    MoveL Offs(pOrigin,403.21,104.24,0.00),v60,z0,tPen\WObj:=wPaper;
    MoveL Offs(pOrigin,403.00,104.66,0.00),v40,z0,tPen\WObj:=wPaper;
    MoveL Offs(pOrigin,403.21,104.24,0.00),v40,fine,tPen\WObj:=wPaper;
    MoveL Offs(pOrigin,403.21,104.24,6.00),v60,z5,tPen\WObj:=wPaper;
    MoveL Offs(pOrigin,397.70,106.78,6.00),vTravel,z5,tPen\WObj:=wPaper;
    MoveL Offs(pOrigin,397.70,106.78,0.00),v60,z0,tPen\WObj:=wPaper;
    MoveL Offs(pOrigin,401.31,110.39,0.00),v40,z0,tPen\WObj:=wPaper;
    MoveL Offs(pOrigin,400.88,110.04,0.00),v40,z0,tPen\WObj:=wPaper;
  ENDPROC

  PROC DrawPart197()
    MoveL Offs(pOrigin,399.60,110.04,0.00),v40,fine,tPen\WObj:=wPaper;
    MoveL Offs(pOrigin,399.60,110.04,6.00),v60,z5,tPen\WObj:=wPaper;
    MoveL Offs(pOrigin,398.31,108.88,6.00),vTravel,z5,tPen\WObj:=wPaper;
    MoveL Offs(pOrigin,398.31,108.88,0.00),v60,z0,tPen\WObj:=wPaper;
    MoveL Offs(pOrigin,396.81,107.38,0.00),v40,z0,tPen\WObj:=wPaper;
    MoveL Offs(pOrigin,396.84,107.93,0.00),v40,z0,tPen\WObj:=wPaper;
    MoveL Offs(pOrigin,398.33,107.93,0.00),v40,fine,tPen\WObj:=wPaper;
    MoveL Offs(pOrigin,398.33,107.93,6.00),v60,z5,tPen\WObj:=wPaper;
    MoveL Offs(pOrigin,397.38,106.15,6.00),vTravel,z5,tPen\WObj:=wPaper;
    MoveL Offs(pOrigin,397.38,106.15,0.00),v60,z0,tPen\WObj:=wPaper;
    MoveL Offs(pOrigin,391.07,112.46,0.00),v40,z0,tPen\WObj:=wPaper;
    MoveL Offs(pOrigin,390.98,112.01,0.00),v40,z0,tPen\WObj:=wPaper;
    MoveL Offs(pOrigin,390.08,111.10,0.00),v40,fine,tPen\WObj:=wPaper;
    MoveL Offs(pOrigin,390.08,111.10,6.00),v60,z5,tPen\WObj:=wPaper;
    MoveL Offs(pOrigin,388.38,107.68,6.00),vTravel,z5,tPen\WObj:=wPaper;
    MoveL Offs(pOrigin,388.38,107.68,0.00),v60,z0,tPen\WObj:=wPaper;
    MoveL Offs(pOrigin,390.79,105.27,0.00),v40,fine,tPen\WObj:=wPaper;
    MoveL Offs(pOrigin,390.79,105.27,6.00),v60,z5,tPen\WObj:=wPaper;
    MoveL Offs(pOrigin,390.93,106.62,6.00),vTravel,z5,tPen\WObj:=wPaper;
    MoveL Offs(pOrigin,390.93,106.62,0.00),v60,z0,tPen\WObj:=wPaper;
    MoveL Offs(pOrigin,392.44,105.12,0.00),v40,fine,tPen\WObj:=wPaper;
    MoveL Offs(pOrigin,392.44,105.12,6.00),v60,z5,tPen\WObj:=wPaper;
    MoveL Offs(pOrigin,394.71,104.66,6.00),vTravel,z5,tPen\WObj:=wPaper;
    MoveL Offs(pOrigin,394.71,104.66,0.00),v60,z0,tPen\WObj:=wPaper;
    MoveL Offs(pOrigin,393.86,104.66,0.00),v40,z0,tPen\WObj:=wPaper;
    MoveL Offs(pOrigin,389.61,106.36,0.00),v40,z0,tPen\WObj:=wPaper;
    MoveL Offs(pOrigin,383.88,107.85,0.00),v40,z0,tPen\WObj:=wPaper;
    MoveL Offs(pOrigin,377.92,108.70,0.00),v40,z0,tPen\WObj:=wPaper;
    MoveL Offs(pOrigin,371.98,108.70,0.00),v40,z0,tPen\WObj:=wPaper;
    MoveL Offs(pOrigin,371.98,108.70,0.00),v40,z0,tPen\WObj:=wPaper;
    MoveL Offs(pOrigin,371.34,108.91,0.00),v40,z0,tPen\WObj:=wPaper;
    MoveL Offs(pOrigin,364.11,107.21,0.00),v40,z0,tPen\WObj:=wPaper;
    MoveL Offs(pOrigin,360.08,105.80,0.00),v40,z0,tPen\WObj:=wPaper;
    MoveL Offs(pOrigin,356.67,104.03,0.00),v40,fine,tPen\WObj:=wPaper;
    MoveL Offs(pOrigin,356.67,104.03,6.00),v60,z5,tPen\WObj:=wPaper;
    MoveL Offs(pOrigin,355.44,104.78,6.00),vTravel,z5,tPen\WObj:=wPaper;
    MoveL Offs(pOrigin,355.44,104.78,0.00),v60,z0,tPen\WObj:=wPaper;
    MoveL Offs(pOrigin,347.47,112.75,0.00),v40,z0,tPen\WObj:=wPaper;
    MoveL Offs(pOrigin,347.54,111.87,0.00),v40,z0,tPen\WObj:=wPaper;
    MoveL Offs(pOrigin,351.44,115.78,0.00),v40,z0,tPen\WObj:=wPaper;
    MoveL Offs(pOrigin,350.94,115.32,0.00),v40,z0,tPen\WObj:=wPaper;
    MoveL Offs(pOrigin,349.02,115.32,0.00),v40,z0,tPen\WObj:=wPaper;
    MoveL Offs(pOrigin,348.45,115.77,0.00),v40,z0,tPen\WObj:=wPaper;
    MoveL Offs(pOrigin,352.96,120.28,0.00),v40,z0,tPen\WObj:=wPaper;
    MoveL Offs(pOrigin,352.85,120.60,0.00),v40,z0,tPen\WObj:=wPaper;
    MoveL Offs(pOrigin,350.09,120.60,0.00),v40,z0,tPen\WObj:=wPaper;
    MoveL Offs(pOrigin,350.30,121.66,0.00),v40,z0,tPen\WObj:=wPaper;
    MoveL Offs(pOrigin,353.28,121.66,0.00),v40,z0,tPen\WObj:=wPaper;
    MoveL Offs(pOrigin,352.72,121.66,0.00),v40,z0,tPen\WObj:=wPaper;
    MoveL Offs(pOrigin,352.72,125.28,0.00),v40,fine,tPen\WObj:=wPaper;
    MoveL Offs(pOrigin,352.72,125.28,6.00),v60,z5,tPen\WObj:=wPaper;
    MoveL Offs(pOrigin,354.31,123.13,6.00),vTravel,z5,tPen\WObj:=wPaper;
    MoveL Offs(pOrigin,354.31,123.13,0.00),v60,z0,tPen\WObj:=wPaper;
    MoveL Offs(pOrigin,348.90,117.72,0.00),v40,z0,tPen\WObj:=wPaper;
    MoveL Offs(pOrigin,348.51,117.69,0.00),v40,z0,tPen\WObj:=wPaper;
    MoveL Offs(pOrigin,355.72,110.47,0.00),v40,z0,tPen\WObj:=wPaper;
    MoveL Offs(pOrigin,354.76,110.61,0.00),v40,z0,tPen\WObj:=wPaper;
    MoveL Offs(pOrigin,355.40,111.25,0.00),v40,z0,tPen\WObj:=wPaper;
    MoveL Offs(pOrigin,354.76,110.61,0.00),v40,z0,tPen\WObj:=wPaper;
    MoveL Offs(pOrigin,354.97,109.73,0.00),v40,z0,tPen\WObj:=wPaper;
    MoveL Offs(pOrigin,348.36,116.34,0.00),v40,fine,tPen\WObj:=wPaper;
    MoveL Offs(pOrigin,348.36,116.34,6.00),v60,z5,tPen\WObj:=wPaper;
    MoveL Offs(pOrigin,348.06,115.14,6.00),vTravel,z5,tPen\WObj:=wPaper;
    MoveL Offs(pOrigin,348.06,115.14,0.00),v60,z0,tPen\WObj:=wPaper;
    MoveL Offs(pOrigin,354.23,108.98,0.00),v40,z0,tPen\WObj:=wPaper;
    MoveL Offs(pOrigin,354.98,108.23,0.00),v40,z0,tPen\WObj:=wPaper;
    MoveL Offs(pOrigin,356.93,106.28,0.00),v40,z0,tPen\WObj:=wPaper;
    MoveL Offs(pOrigin,356.25,106.87,0.00),v40,z0,tPen\WObj:=wPaper;
    MoveL Offs(pOrigin,354.76,106.87,0.00),v40,z0,tPen\WObj:=wPaper;
    MoveL Offs(pOrigin,354.76,107.21,0.00),v40,z0,tPen\WObj:=wPaper;
    MoveL Offs(pOrigin,355.40,107.64,0.00),v40,z0,tPen\WObj:=wPaper;
    MoveL Offs(pOrigin,354.76,107.21,0.00),v40,fine,tPen\WObj:=wPaper;
    MoveL Offs(pOrigin,354.76,107.21,6.00),v60,z5,tPen\WObj:=wPaper;
    MoveL Offs(pOrigin,354.98,105.82,6.00),vTravel,z5,tPen\WObj:=wPaper;
    MoveL Offs(pOrigin,354.98,105.82,0.00),v60,z0,tPen\WObj:=wPaper;
    MoveL Offs(pOrigin,353.49,105.82,0.00),v40,z0,tPen\WObj:=wPaper;
    MoveL Offs(pOrigin,353.06,105.72,0.00),v40,z0,tPen\WObj:=wPaper;
    MoveL Offs(pOrigin,353.70,106.36,0.00),v40,z0,tPen\WObj:=wPaper;
    MoveL Offs(pOrigin,353.06,105.72,0.00),v40,z0,tPen\WObj:=wPaper;
    MoveL Offs(pOrigin,353.49,104.66,0.00),v40,z0,tPen\WObj:=wPaper;
    MoveL Offs(pOrigin,354.34,105.51,0.00),v40,z0,tPen\WObj:=wPaper;
    MoveL Offs(pOrigin,353.49,104.66,0.00),v40,z0,tPen\WObj:=wPaper;
    MoveL Offs(pOrigin,353.64,103.59,0.00),v40,z0,tPen\WObj:=wPaper;
    MoveL Offs(pOrigin,346.88,110.35,0.00),v40,fine,tPen\WObj:=wPaper;
    MoveL Offs(pOrigin,346.88,110.35,6.00),v60,z5,tPen\WObj:=wPaper;
    MoveL Offs(pOrigin,346.14,108.11,6.00),vTravel,z5,tPen\WObj:=wPaper;
    MoveL Offs(pOrigin,346.14,108.11,0.00),v60,z0,tPen\WObj:=wPaper;
    MoveL Offs(pOrigin,352.15,102.10,0.00),v40,fine,tPen\WObj:=wPaper;
    MoveL Offs(pOrigin,352.15,102.10,6.00),v60,z5,tPen\WObj:=wPaper;
    MoveL Offs(pOrigin,354.76,105.72,6.00),vTravel,z5,tPen\WObj:=wPaper;
    MoveL Offs(pOrigin,354.76,105.72,0.00),v60,z0,tPen\WObj:=wPaper;
    MoveL Offs(pOrigin,355.40,106.36,0.00),v40,z0,tPen\WObj:=wPaper;
    MoveL Offs(pOrigin,354.76,105.72,0.00),v40,fine,tPen\WObj:=wPaper;
    MoveL Offs(pOrigin,354.76,105.72,6.00),v60,z5,tPen\WObj:=wPaper;
    MoveL Offs(pOrigin,356.18,105.53,6.00),vTravel,z5,tPen\WObj:=wPaper;
    MoveL Offs(pOrigin,356.18,105.53,0.00),v60,z0,tPen\WObj:=wPaper;
    MoveL Offs(pOrigin,347.77,113.94,0.00),v40,z0,tPen\WObj:=wPaper;
    MoveL Offs(pOrigin,347.99,113.82,0.00),v40,z0,tPen\WObj:=wPaper;
    MoveL Offs(pOrigin,351.90,117.73,0.00),v40,z0,tPen\WObj:=wPaper;
    MoveL Offs(pOrigin,351.58,117.43,0.00),v40,z0,tPen\WObj:=wPaper;
    MoveL Offs(pOrigin,349.45,117.43,0.00),v40,fine,tPen\WObj:=wPaper;
    MoveL Offs(pOrigin,349.45,117.43,6.00),v60,z5,tPen\WObj:=wPaper;
    MoveL Offs(pOrigin,348.81,114.26,6.00),vTravel,z5,tPen\WObj:=wPaper;
    MoveL Offs(pOrigin,348.81,114.26,0.00),v60,z0,tPen\WObj:=wPaper;
    MoveL Offs(pOrigin,350.94,114.26,0.00),v40,z0,tPen\WObj:=wPaper;
    MoveL Offs(pOrigin,350.72,113.21,0.00),v40,z0,tPen\WObj:=wPaper;
    MoveL Offs(pOrigin,348.60,113.21,0.00),v40,fine,tPen\WObj:=wPaper;
    MoveL Offs(pOrigin,348.60,113.21,6.00),v60,z5,tPen\WObj:=wPaper;
    MoveL Offs(pOrigin,350.61,109.98,6.00),vTravel,z5,tPen\WObj:=wPaper;
    MoveL Offs(pOrigin,350.61,109.98,0.00),v60,z0,tPen\WObj:=wPaper;
    MoveL Offs(pOrigin,350.61,107.21,0.00),v40,z0,tPen\WObj:=wPaper;
    MoveL Offs(pOrigin,351.15,107.21,0.00),v40,z0,tPen\WObj:=wPaper;
    MoveL Offs(pOrigin,351.58,107.64,0.00),v40,z0,tPen\WObj:=wPaper;
    MoveL Offs(pOrigin,351.15,107.21,0.00),v40,z0,tPen\WObj:=wPaper;
    MoveL Offs(pOrigin,351.15,106.87,0.00),v40,z0,tPen\WObj:=wPaper;
    MoveL Offs(pOrigin,346.69,106.87,0.00),v40,fine,tPen\WObj:=wPaper;
    MoveL Offs(pOrigin,346.69,106.87,6.00),v60,z5,tPen\WObj:=wPaper;
    MoveL Offs(pOrigin,344.36,102.42,6.00),vTravel,z5,tPen\WObj:=wPaper;
    MoveL Offs(pOrigin,344.36,102.42,0.00),v60,z0,tPen\WObj:=wPaper;
    MoveL Offs(pOrigin,350.82,95.96,0.00),v40,z0,tPen\WObj:=wPaper;
  ENDPROC

